// TwinCAT 3 PLC project TFM
// ProgramVersion: 3.1.4024.0
// libraries:
//   Tc2_Standard, * (Beckhoff Automation GmbH)
//   Tc2_System, * (Beckhoff Automation GmbH)
//   Tc2_Utilities, * (Beckhoff Automation GmbH)
//   Tc3_Module, * (Beckhoff Automation GmbH)
//   VisuDialogs, * (System)
//   VisuSymbols,3.5.10.0,System
// project tree:
//   DUTs/ DUT_Guardado_Almacen.TcDUT (not stored), DUT_Input.TcDUT
//   / GlobalTextList.TcGTLO, PlcTask.TcTTO (not stored), Visualization Manager.TcVMO (not stored)
//   GVLs/ GVL.TcGVL
//   POUs/Almacén/ FB_Visibilidad.TcPOU (not stored), FUN_get_Posicion_Libre_Array.TcPOU (not stored), FUN_get_Posicion_Ocupada_Array.TcPOU, POU_Almacen.TcPOU, POU_Cruce_Almacen.TcPOU, POU_Linea_Almacen.TcPOU
//   POUs/Control funcionalidad/ Contadores_Control_Lineas.TcPOU, FB_Control_Estacion.TcPOU, POU_Control_Estaciones.TcPOU (not stored), POU_Edges.TcPOU, POU_Parada.TcPOU (not stored), POU_Reset_Planta.TcPOU
//   POUs/Entrada y división/ Etapa1.TcPOU
//   POUs/Línea producción/ Linea_Produccion.TcPOU (not stored), POU_Pinzas.TcPOU
//   POUs/ MAIN.TcPOU (not stored)
//   POUs/Módulos/ POU_Control_Planta_1.TcPOU (not stored), POU_Funcionamiento.TcPOU (not stored), POU_Mando.TcPOU, POU_Seguridad.TcPOU
//   VISUs/Manual/ Almacen_Manual.TcVIS, Entrada_Manual.TcVIS (not stored), Linea_Almacen_Manual.TcVIS, Linea_Produccion_Azul_1.TcVIS, Linea_Produccion_Azul_2.TcVIS
//   VISUs/ Pantalla_Principal.TcVIS (not stored), HMI.TcVIS
// real-time tasks:
//   TASK PlcTask: cycle T#10ms, priority 20, ADS port 350

// ---- DUTs/DUT_Input.TcDUT
TYPE DUT_Input :
STRUCT
	Max_Capas_Apiladas_Azul  : INT := 2; 	  // Cantidad de capas a apilar en el paletizador	
	Max_Capas_Apiladas_Verde : INT := 2;	  // Cantidad de capas a apilar en el paletizador	
	Max_Capas_Apiladas_Metal : INT := 2; 	  // Cantidad de capas a apilar en el paletizador
	Descartar_Pieza_Azul 	 : BOOL := FALSE; // Control de ingreso de material a la línea Azul
	Descartar_Pieza_Verde  	 : BOOL := FALSE; // Control de ingreso de material a la línea Verde
	Descartar_Pieza_Metal 	 : BOOL := FALSE; // Control de ingreso de material a la línea Metal
END_STRUCT
END_TYPE

// ---- GVLs/GVL.TcGVL
//{attribute 'qualified_only'}
VAR_GLOBAL

// LOCAL
	
	Manual : BOOL := FALSE; // Control modo manual/automático
	Marcha : BOOL := FALSE; // Control modo de operación de la planta
	
	//CONTADORES TOTALES PARA BASE DE DATOS
	
	Contador_Totales_Azul_Separadas 	 : INT := 0;  // Piezas totales azules pasadas a la linea de produccion
	Contador_Totales_Verde_Separadas 	 : INT := 0;  // Piezas totales verdes pasadas a la linea de producción
	Contador_Totales_Metal_Separadas 	 : INT := 0;  // Piezas totales metalicas pasadas a la linea de producción
	Contador_Piezas_Totales_Emitidas 	 : INT := 0;  // Piezas totales emitidas por el emisor
	Contador_Piezas_Totales_Descartadas  : INT := 0;  // Piezas totales descartadas
	Contador_Palets_Azules_Totales  	 : INT := 0;  // Palets de productos azules completados
	Contador_Palets_Verdes_Totales  	 : INT := 0;  // Palets de productos verdes completados
	Contador_Palets_Metales_Totales 	 : INT := 0;  // Palets de productos metales completados
	Pallets_Almacenados 				 : DINT := 0; // Cantidad de palets almacenados sin contar los extraidos
	Pallets_Almacenados_Retirados		 : DINT := 0; // Totalidad de palets extraidos
	Pallets_Azules_Totales_Emitidos  	 : DINT := 0; // Cantidad de palets emitidos para ser "rellenados", esta variable se usa para controlar los errores del RFID		
	Pallets_Verdes_Totales_Emitidos   	 : DINT := 0; // Cantidad de palets emitidos para ser "rellenados", esta variable se usa para controlar los errores del RFID	
	Pallets_Metalicos_Totales_Emitidos   : DINT := 0; // Cantidad de palets emitidos para ser "rellenados", esta variable se usa para controlar los errores del RFID	
	
	// CONTADORES-FLAGS PARA CONTROL DE LINEA	

	//Contador_Piezas_No_Descartadas : INT := 0; // Piezas utilizables emitidas por el emitter 1,
	Capas_Apiladas_Azul					 : INT := 0;  // Capas de cajas de producto azul apiladas en el palet
	Capas_Apiladas_Metal				 : INT := 0;  // Capas de cajas de producto verde apiladas en el palet
	Capas_Apiladas_Verde				 : INT := 0;  // Capas de cajas de producto metálico apiladas en el palet
	Contador_Piezas_Zona_Pivot_Principal : INT := 0;  // Piezas en la zona Pivot y descarte
	Contador_Pivot_Azul 				 : INT := 0;  // Piezas en la zona Pivot de la linea azul
	Contador_Pivot_Verde 				 : INT := 0;  // Piezas en la zona Pivot de la linea verde
	Contador_Pivot_Metal 				 : INT := 0;  // Piezas en la zona Pivot de la linea metal
	Contador_Manipulador_1 				 : INT := 0;  // Piezas que hay dentro de la celda del robot
	Contador_Manipulador_2				 : INT := 0;  // Piezas que hay dentro de la celda del robot
	Contador_Manipulador_3				 : INT := 0;  // Piezas que hay dentro de la celda del robot
	Contador_Manipulador_4				 : INT := 0;  // Piezas que hay dentro de la celda del robot
	Contador_Manipulador_5				 : INT := 0;  // Piezas que hay dentro de la celda del robot
	Contador_Manipulador_6				 : INT := 0;  // Piezas que hay dentro de la celda del robot
	Contador_Linea_Manipulador_1_I		 : INT := 0;  // Piezas que hay en la cinta de entrada al manipulador
	Contador_Linea_Manipulador_2_I		 : INT := 0;  // Piezas que hay en la cinta de entrada al manipulador
	Contador_Linea_Manipulador_3_I		 : INT := 0;  // Piezas que hay en la cinta de entrada al manipulador	
	Contador_Linea_Manipulador_4_I		 : INT := 0;  // Piezas que hay en la cinta de entrada al manipulador	
	Contador_Linea_Manipulador_5_I		 : INT := 0;  // Piezas que hay en la cinta de entrada al manipulador
	Contador_Linea_Manipulador_6_I		 : INT := 0;  // Piezas que hay en la cinta de entrada al manipulador	
	Contador_Linea_Principal			 : INT := 0;  // Elementos en la línea principal de entrada tras el sensor de visión
	Contador_Manipulador_1_Lid			 : INT := 0;  // Piezas que hay en la cinta de salida del manipulador	
	Contador_Manipulador_2_Lid			 : INT := 0;  // Piezas que hay en la cinta de salida del manipulador	
	Contador_Manipulador_3_Lid			 : INT := 0;  // Piezas que hay en la cinta de salida del manipulador
	Contador_Manipulador_1_Base			 : INT := 0;  // Piezas que hay en la cinta de salida del manipulador
	Contador_Manipulador_2_Base			 : INT := 0;  // Piezas que hay en la cinta de salida del manipulador
	Contador_Manipulador_3_Base 		 : INT := 0;  // Piezas que hay en la cinta de salida del manipulador
	Contador_Box_Azul					 : INT := 0;  // Cajas de producto azul entrando al paletizado
	Contador_Box_Verde					 : INT := 0;  // Cajas de producto verde entrando al paletizado
	Contador_Box_Metal 					 : INT := 0;  // Cajas de producto metálico entrando al paletizado
	Contador_Palets_Azules   			 : INT := 0;  // Palets de producto azul en el primer tramo de rodillos	
	Contador_Palets_Verdes				 : INT := 0;  // Palets de producto verde en el primer tramo de rodillos	
	Contador_Palets_Metal				 : INT := 0;  // Palets de producto metálico en el primer tramo de rodillos
	Contador_Linea_Cruce_1				 : INT := 0;  // Palets que hay entre los dos cruces de rodillos
	Contador_Linea_Cruce_2				 : INT := 0;  // Palets entre el último cruce y el almacen	
	Linea_Salida_Libre_2				 : BOOL := TRUE; // Control de cinta de salida para el paletizado de laínea verde, si la línea de salida no está libre, no puede sacar el palet
	Linea_Salida_Libre_3				 : BOOL := TRUE; // Control de cinta de salida para el paletizado de la línea metálica, si la línea de salida no está libre, no puede sacar el palet

	// VARIABLES PARA CONTROLAR ACCIONES	
	
	Sacar_Palet_1 			: BOOL := FALSE; // Para saber si el palet de producto azul del paletizador tiene via libre para ser pasado a los rodillos camino al almacen
	Sacar_Palet_2 			: BOOL := FALSE; // Para saber si el palet de producto verde del paletizador tiene via libre para ser pasado a los rodillos camino al almacen
	Sacar_Palet_3			: BOOL := FALSE; // Para saber si el palet de producto metálico  paletizador tiene via libre para ser pasado a los rodillos camino al almacen
	Error_RFID_1 			: BOOL := FALSE; // Variable que guarda si ha habido error a la hora de escribir información en un palet en la línea azul	
	Error_RFID_2 			: BOOL := FALSE; // Variable que guarda si ha habido error a la hora de escribir información en un palet en la línea verde
	Error_RFID_3 			: BOOL := FALSE; // Variable que guarda si ha habido error a la hora de escribir información en un palet en la línea metálica
	Error_RFID_Almacen 		: BOOL := FALSE; // Variable que guarda si ha habido error a la hora de leer información en un palet a almacenar
	Control_TAPP_A 			: BOOL := FALSE; // En base a la botonera de control y los sensores de puerta, se permite el movimiento o no del Pick&Place de la línea azul
	Control_TAPP_V 			: BOOL := FALSE; // En base a la botonera de control y los sensores de puerta, se permite el movimiento o no del Pick&Place de la línea verde
	Control_TAPP_M 			: BOOL := FALSE; // En base a la botonera de control y los sensores de puerta, se permite el movimiento o no del Pick&Place de la línea metálica
	Control_Paletizador_A 	: BOOL := FALSE; // En base a la botonera de control y los sensores de puerta, se permite el movimiento o no del paletizador de la línea azul
	Control_Paletizador_V 	: BOOL := FALSE; // En base a la botonera de control y los sensores de puerta, se permite el movimiento o no del paletizador de la línea verde
	Control_Paletizador_M 	: BOOL := FALSE; // En base a la botonera de control y los sensores de puerta, se permite el movimiento o no del paletizador de la línea metálica
	Control_Almacen 		: BOOL := FALSE; // En base a la botonera de control y los sensores de puerta, se permite el movimiento o no de la grúa del alamcén
	Reset					: BOOL := FALSE; // Variable para resetear los contadores
	
	//ESTADOS	
	Estado_Pick_Place_1 	: INT  := 0; // Estado del Pick&Place de la línea azul
	Estado_Palletizer_1 	: INT  := 0; // Estado del Pick&Place de la línea verde
	Estado_Pick_Place_2 	: INT  := 0; // Estado del Pick&Place de la línea metálica
	Estado_Palletizer_2 	: INT  := 0; // Estado del paletizador de la línea azul
	Estado_Pick_Place_3 	: INT  := 0; // Estado del paletizador de la línea verde
	Estado_Palletizer_3 	: INT  := 0; // Estado del paletizador de la línea metálica	
	Estado_Almacen_I 		: INT  := 0; // Estado de la grúa en modo almacenamiento
	Estado_Almacen_O 		: INT  := 1; // Estado de la grúa en modo extracción
	
	// ALMACEN
	
	ContadorPalets			: INT := 0; 							// Contador de palets del Almacen en base a la selección del display
	Retirada_Start			: BOOL := FALSE; 						// Guarda la pulsación del botón start para extraer del almacen
	Clasificados 			: ARRAY[0..53] OF DUT_Guardado_Almacen; // Estanteria: 0 (posicion libre), 1 (id blue raw material), 4 (id green raw material), 7 (id metal raw material)
	Input					: ARRAY[0..0] OF DUT_Input; 			// Variables de entrada para controlar la funcionalidad del flujo.

// --------------------------- ENTRADAS ---------------------------

// Etapa Entrada 

	{attribute 'OPC.UA.DA' := '1'}
	Diffuse_Sensor_0 AT %I* : BOOL;
	{attribute 'OPC.UA.DA' := '1'}
	Diffuse_Sensor_1 AT %I* : BOOL;
	{attribute 'OPC.UA.DA' := '1'} 
	Diffuse_Sensor_2 AT %I* : BOOL;
	{attribute 'OPC.UA.DA' := '1'} 
	Diffuse_Sensor_3 AT %I* : BOOL;
	{attribute 'OPC.UA.DA' := '1'} 
	Diffuse_Sensor_4 AT %I* : BOOL;
	{attribute 'OPC.UA.DA' := '1'} 
	Diffuse_Sensor_5 AT %I* : BOOL;
	{attribute 'OPC.UA.DA' := '1'} 
	Diffuse_Sensor_8 AT %I* : BOOL;
	{attribute 'OPC.UA.DA' := '1'} 
	Diffuse_Sensor_9 AT %I* : BOOL;
	{attribute 'OPC.UA.DA' := '1'} 
	Diffuse_Sensor_12 AT %I* : BOOL;
	{attribute 'OPC.UA.DA' := '1'} 
	Emergency_Stop_2 AT %I* : BOOL;
	{attribute 'OPC.UA.DA' := '1'} 	
	Pusher_1_Front_Limit AT %I* : BOOL;
	{attribute 'OPC.UA.DA' := '1'} 
	Pusher_2_Front_Limit AT %I* : BOOL;
	{attribute 'OPC.UA.DA' := '1'} 
	Pusher_3_Front_Limit AT %I* : BOOL;	
	{attribute 'OPC.UA.DA' := '1'} 
	Reset_Button_2: BOOL;
	{attribute 'OPC.UA.DA' := '1'} 
	Start_Button_2 AT %I* : BOOL;
	{attribute 'OPC.UA.DA' := '1'} 
	Stop_Button_2 AT %I* : BOOL;
	

// Linea Producción 1 
	
	{attribute 'OPC.UA.DA' := '1'} 
	Diffuse_Sensor_15 AT %I* : BOOL;
	{attribute 'OPC.UA.DA' := '1'} 
	Diffuse_Sensor_16 AT %I* : BOOL;	
	{attribute 'OPC.UA.DA' := '1'} 
	Diffuse_Sensor_45 AT %I* : BOOL;
	{attribute 'OPC.UA.DA' := '1'} 
	Diffuse_Sensor_46 AT %I* : BOOL;
	{attribute 'OPC.UA.DA' := '1'} 
	Emergency_Stop_3 AT %I* : BOOL;
	{attribute 'OPC.UA.DA' := '1'}
	Emergency_Stop_4 AT %I* : BOOL;
	//{attribute 'OPC.UA.DA' := '1'} 
	Reset_Button_3 AT %I* : BOOL;
	//{attribute 'OPC.UA.DA' := '1'} 
	Reset_Button_4 AT %I* : BOOL;	
	//{attribute 'OPC.UA.DA' := '1'} 
	Safety_Door_1 AT %I* : BOOL;
	//{attribute 'OPC.UA.DA' := '1'} 
	Safety_Door_2 AT %I* : BOOL;
	//{attribute 'OPC.UA.DA' := '1'} 
	Safety_Door_3 AT %I* : BOOL;
	//{attribute 'OPC.UA.DA' := '1'} 
	Safety_Door_4 AT %I* : BOOL;
	//{attribute 'OPC.UA.DA' := '1'} 
	Start_Button_3 AT %I* : BOOL;
	//{attribute 'OPC.UA.DA' := '1'} 
	Stop_Button_3 AT %I* : BOOL;
	//{attribute 'OPC.UA.DA' := '1'} //Comentar
	Start_Button_6 AT %I* : BOOL;
	//{attribute 'OPC.UA.DA' := '1'} //Comentar
	Stop_Button_6 AT %I* : BOOL;
	
	
	//Función
	
	{attribute 'OPC.UA.DA' := '1'} 
	Diffuse_Sensor_6 AT %I* : BOOL;
	{attribute 'OPC.UA.DA' := '1'} 
	Diffuse_Sensor_7 AT %I* : BOOL;
	{attribute 'OPC.UA.DA' := '1'} 
	Diffuse_Sensor_17 AT %I* : BOOL;	
	{attribute 'OPC.UA.DA' := '1'} 
	Diffuse_Sensor_18 AT %I* : BOOL;	
	{attribute 'OPC.UA.DA' := '1'} 
	Diffuse_Sensor_19 AT %I* : BOOL;	
	{attribute 'OPC.UA.DA' := '1'} 
	Diffuse_Sensor_20 AT %I* : BOOL;
	{attribute 'OPC.UA.DA' := '1'} 
	Diffuse_Sensor_21 AT %I* : BOOL;
	{attribute 'OPC.UA.DA' := '1'} 
	Diffuse_Sensor_22 AT %I* : BOOL;
	{attribute 'OPC.UA.DA' := '1'}  // Comentar
	Palletizer_1_Clamped AT %I* : BOOL;	
	{attribute 'OPC.UA.DA' := '1'}  // Comentar
	Palletizer_1_Plate_Limit AT %I* : BOOL;	
	{attribute 'OPC.UA.DA' := '1'}  // Comentar
	Palletizer_1_Pusher_Limit AT %I* : BOOL;
	{attribute 'OPC.UA.DA' := '1'}  // Comentar
	Palletizer_1_Elevator_Back_Limit AT %I* : BOOL;	
	{attribute 'OPC.UA.DA' := '1'}  // Comentar
	Palletizer_1_Elevator_Front_Limit AT %I* : BOOL;	
	{attribute 'OPC.UA.DA' := '1'}  // Comentar
	Palletizer_1_Elevator_Moving AT %I* : BOOL;	
	{attribute 'OPC.UA.DA' := '1'}  // Comentar
	RFID_Reader_1_Status AT %I* : DINT;	
	{attribute 'OPC.UA.DA' := '1'}  // Comentar
	RFID_Reader_1_Command_ID AT %I* : DINT;	
	//{attribute 'OPC.UA.DA' := '1'} 
	Right_Positioner_1_Clamped AT %I* : BOOL;
	{attribute 'OPC.UA.DA' := '1'}  // Comentar
	Right_Positioner_2_Clamped AT %I* : BOOL;
	{attribute 'OPC.UA.DA' := '1'}  // Comentar
	Right_Positioner_2_Limit AT %I* : BOOL;	
	{attribute 'OPC.UA.DA' := '1'}  // Comentar
	Two_Axis_Pick_Place_1_Detected AT %I* : BOOL;	
	{attribute 'OPC.UA.DA' := '1'}  // Comentar
	Two_Axis_Pick_Place_1_MovingX AT %I* : BOOL;
	{attribute 'OPC.UA.DA' := '1'}  // Comentar
	Two_Axis_Pick_Place_1_MovingZ AT %I* : BOOL;
	
	
// Línea Producción 2	
	
	{attribute 'OPC.UA.DA' := '1'} 
	Diffuse_Sensor_23 AT %I* : BOOL;
	{attribute 'OPC.UA.DA' := '1'} 
	Diffuse_Sensor_24 AT %I* : BOOL;
	{attribute 'OPC.UA.DA' := '1'} 
	Diffuse_Sensor_47 AT %I* : BOOL;
	{attribute 'OPC.UA.DA' := '1'} 
	Diffuse_Sensor_48 AT %I* : BOOL;
	{attribute 'OPC.UA.DA' := '1'}
	Emergency_Stop_5 AT %I* : BOOL;
	{attribute 'OPC.UA.DA' := '1'}
	Emergency_Stop_6 AT %I* : BOOL;
	//{attribute 'OPC.UA.DA' := '1'} 
	Reset_Button_5 AT %I* : BOOL;
	{attribute 'OPC.UA.DA' := '1'} 
	Reset_Button_6 AT %I* : BOOL;
	//{attribute 'OPC.UA.DA' := '1'} //Comentar
	Safety_Door_5 AT %I* : BOOL;
	//{attribute 'OPC.UA.DA' := '1'} //Comentar
	Safety_Door_6 AT %I* : BOOL;
	//{attribute 'OPC.UA.DA' := '1'} //Comentar
	Safety_Door_7 AT %I* : BOOL;
	//{attribute 'OPC.UA.DA' := '1'} //Comentar
	Safety_Door_8 AT %I* : BOOL;
	//{attribute 'OPC.UA.DA' := '1'} 
	Start_Button_4 AT %I* : BOOL;
	//{attribute 'OPC.UA.DA' := '1'} 
	Stop_Button_4 AT %I* : BOOL;
	//{attribute 'OPC.UA.DA' := '1'} //Comentar
	Start_Button_7 AT %I* : BOOL;
	//{attribute 'OPC.UA.DA' := '1'} //Comentar
	Stop_Button_7 AT %I* : BOOL;
	
	
	//Función
	
	{attribute 'OPC.UA.DA' := '1'} 
	Diffuse_Sensor_10 AT %I* : BOOL;
	{attribute 'OPC.UA.DA' := '1'} 
	Diffuse_Sensor_11 AT %I* : BOOL;
	{attribute 'OPC.UA.DA' := '1'} 
	Diffuse_Sensor_25 AT %I* : BOOL;
	{attribute 'OPC.UA.DA' := '1'} 
	Diffuse_Sensor_26 AT %I* : BOOL;
	{attribute 'OPC.UA.DA' := '1'} 
	Diffuse_Sensor_27 AT %I* : BOOL;
	{attribute 'OPC.UA.DA' := '1'} 
	Diffuse_Sensor_28 AT %I* : BOOL;
	{attribute 'OPC.UA.DA' := '1'} 
	Diffuse_Sensor_29 AT %I* : BOOL;
	{attribute 'OPC.UA.DA' := '1'} 
	Diffuse_Sensor_30 AT %I* : BOOL;
	//{attribute 'OPC.UA.DA' := '1'} // Comentar
	Palletizer_2_Clamped AT %I* : BOOL;	
	//{attribute 'OPC.UA.DA' := '1'}  // Comentar
	Palletizer_2_Plate_Limit AT %I* : BOOL;	
	//{attribute 'OPC.UA.DA' := '1'}  // Comentar
	Palletizer_2_Pusher_Limit AT %I* : BOOL;
	//{attribute 'OPC.UA.DA' := '1'}  // Comentar
	Palletizer_2_Elevator_Back_Limit AT %I* : BOOL;	
	//{attribute 'OPC.UA.DA' := '1'}  // Comentar
	Palletizer_2_Elevator_Front_Limit AT %I* : BOOL;	
	//{attribute 'OPC.UA.DA' := '1'}  // Comentar
	Palletizer_2_Elevator_Moving AT %I* : BOOL;
	//{attribute 'OPC.UA.DA' := '1'}  // Comentar
	RFID_Reader_2_Status AT %I* : DINT;	
	//{attribute 'OPC.UA.DA' := '1'}
	RFID_Reader_2_Command_ID AT %I* : DINT;
	//{attribute 'OPC.UA.DA' := '1'}  // Comentar
	Right_Positioner_3_Clamped AT %I* : BOOL;	
	//{attribute 'OPC.UA.DA' := '1'}  // Comentar
	Right_Positioner_4_Clamped AT %I* : BOOL;
	//{attribute 'OPC.UA.DA' := '1'}  // Comentar
	Right_Positioner_4_Limit AT %I* : BOOL;
	//{attribute 'OPC.UA.DA' := '1'}  // Comentar
	Two_Axis_Pick_Place_2_Detected AT %I* : BOOL;
	//{attribute 'OPC.UA.DA' := '1'}  // Comentar
	Two_Axis_Pick_Place_2_MovingX AT %I* : BOOL;
	//{attribute 'OPC.UA.DA' := '1'}  // Comentar
	Two_Axis_Pick_Place_2_MovingZ AT %I* : BOOL;
	

// Línea Producción 3

	{attribute 'OPC.UA.DA' := '1'} 
	Diffuse_Sensor_31 AT %I* : BOOL;
	{attribute 'OPC.UA.DA' := '1'} 
	Diffuse_Sensor_32 AT %I* : BOOL;
	{attribute 'OPC.UA.DA' := '1'} 
	Diffuse_Sensor_49 AT %I* : BOOL;
	{attribute 'OPC.UA.DA' := '1'} 
	Diffuse_Sensor_50 AT %I* : BOOL;	
	{attribute 'OPC.UA.DA' := '1'}
	Emergency_Stop_7 AT %I* : BOOL;
	{attribute 'OPC.UA.DA' := '1'}
	Emergency_Stop_8 AT %I* : BOOL;
	//{attribute 'OPC.UA.DA' := '1'} 
	Reset_Button_7 AT %I* : BOOL;
	//{attribute 'OPC.UA.DA' := '1'} 
	Reset_Button_8 AT %I* : BOOL;
	//{attribute 'OPC.UA.DA' := '1'} //Comentar
	Safety_Door_9 AT %I* : BOOL;
	//{attribute 'OPC.UA.DA' := '1'} //Comentar
	Safety_Door_10 AT %I* : BOOL;
	//{attribute 'OPC.UA.DA' := '1'} //Comentar
	Safety_Door_11 AT %I* : BOOL;
	//{attribute 'OPC.UA.DA' := '1'} //Comentar
	Safety_Door_12 AT %I* : BOOL;
	//{attribute 'OPC.UA.DA' := '1'} //Comentar
	Start_Button_5 AT %I* : BOOL;
	//{attribute 'OPC.UA.DA' := '1'} //Comentar
	Stop_Button_5 AT %I* : BOOL;
	//{attribute 'OPC.UA.DA' := '1'} //Comentar
	Start_Button_8 AT %I* : BOOL;
	//{attribute 'OPC.UA.DA' := '1'} //Comentar
	Stop_Button_8 AT %I* : BOOL;
	
	
	//Función
	
	{attribute 'OPC.UA.DA' := '1'} 
	Diffuse_Sensor_13 AT %I* : BOOL;
	{attribute 'OPC.UA.DA' := '1'} 
	Diffuse_Sensor_14 AT %I* : BOOL;
	{attribute 'OPC.UA.DA' := '1'} 
	Diffuse_Sensor_33 AT %I* : BOOL;
	{attribute 'OPC.UA.DA' := '1'} 
	Diffuse_Sensor_34 AT %I* : BOOL;
	{attribute 'OPC.UA.DA' := '1'} 
	Diffuse_Sensor_35 AT %I* : BOOL;
	{attribute 'OPC.UA.DA' := '1'} 
	Diffuse_Sensor_36 AT %I* : BOOL;
	{attribute 'OPC.UA.DA' := '1'} 
	Diffuse_Sensor_37 AT %I* : BOOL;
	{attribute 'OPC.UA.DA' := '1'} 
	Diffuse_Sensor_38 AT %I* : BOOL;
	//{attribute 'OPC.UA.DA' := '1'}  // Comentar
	Palletizer_3_Clamped AT %I* : BOOL;	
	//{attribute 'OPC.UA.DA' := '1'}  // Comentar
	Palletizer_3_Plate_Limit AT %I* : BOOL;
	//{attribute 'OPC.UA.DA' := '1'}  // Comentar
	Palletizer_3_Pusher_Limit AT %I* : BOOL;
	//{attribute 'OPC.UA.DA' := '1'}  // Comentar
	Palletizer_3_Elevator_Back_Limit AT %I* : BOOL;
	//{attribute 'OPC.UA.DA' := '1'}  // Comentar
	Palletizer_3_Elevator_Front_Limit AT %I* : BOOL;
	//{attribute 'OPC.UA.DA' := '1'}  // Comentar
	Palletizer_3_Elevator_Moving AT %I* : BOOL;	
	//{attribute 'OPC.UA.DA' := '1'}  // Comentar
	RFID_Reader_3_Status AT %I* : DINT;	
	//{attribute 'OPC.UA.DA' := '1'}  // Comentar
	RFID_Reader_3_Command_ID AT %I* : DINT;	
	//{attribute 'OPC.UA.DA' := '1'}  // Comentar
	Right_Positioner_5_Clamped AT %I* : BOOL;
	//{attribute 'OPC.UA.DA' := '1'}  // Comentar
	Right_Positioner_6_Clamped AT %I* : BOOL;
	//{attribute 'OPC.UA.DA' := '1'}  // Comentar
	Right_Positioner_6_Limit AT %I* : BOOL;
	//{attribute 'OPC.UA.DA' := '1'}  // Comentar
	Two_Axis_Pick_Place_3_Detected AT %I* : BOOL;
	//{attribute 'OPC.UA.DA' := '1'}  // Comentar
	Two_Axis_Pick_Place_3_MovingX AT %I* : BOOL;
	//{attribute 'OPC.UA.DA' := '1'}  // Comentar
	Two_Axis_Pick_Place_3_MovingZ AT %I* : BOOL;
	
	
//Línea Almacén
	
	{attribute 'OPC.UA.DA' := '1'} 
	Diffuse_Sensor_39 AT %I* : BOOL;
	{attribute 'OPC.UA.DA' := '1'} 
	Diffuse_Sensor_40 AT %I* : BOOL;
	{attribute 'OPC.UA.DA' := '1'} 
	Diffuse_Sensor_41 AT %I* : BOOL;
	{attribute 'OPC.UA.DA' := '1'} 
	Diffuse_Sensor_42 AT %I* : BOOL;
	{attribute 'OPC.UA.DA' := '1'} 
	Diffuse_Sensor_43 AT %I* : BOOL;
	{attribute 'OPC.UA.DA' := '1'} 
	Diffuse_Sensor_44 AT %I* : BOOL;
	{attribute 'OPC.UA.DA' := '1'} 
	Emergency_Stop_1 AT %I* : BOOL;
	{attribute 'OPC.UA.DA' := '1'}
	Emergency_Stop_9 AT %I* : BOOL;
	{attribute 'OPC.UA.DA' := '1'} 
	Stacker_Crane_1_Left_Limit AT %I* : BOOL;	
	{attribute 'OPC.UA.DA' := '1'} 
	Stacker_Crane_1_Middle_Limit AT %I* : BOOL;
	{attribute 'OPC.UA.DA' := '1'} 
	Stacker_Crane_1_Moving_X AT %I* : BOOL;
	{attribute 'OPC.UA.DA' := '1'} 
	Stacker_Crane_1_Moving_Z AT %I* : BOOL;
	{attribute 'OPC.UA.DA' := '1'} 
	Stacker_Crane_1_Right_Limit AT %I* : BOOL;
	{attribute 'OPC.UA.DA' := '1'} 
	Turnable_1_Back_Limit AT %I* : BOOL;
	{attribute 'OPC.UA.DA' := '1'} 
	Turnable_1_Limit_0 AT %I* : BOOL;
	{attribute 'OPC.UA.DA' := '1'} 
	Turnable_1_Limit_90 AT %I* : BOOL;
	{attribute 'OPC.UA.DA' := '1'} 
	Turnable_2_Back_Limit AT %I* : BOOL;
	{attribute 'OPC.UA.DA' := '1'} 
	Turnable_2_Limit_0 AT %I* : BOOL;
	{attribute 'OPC.UA.DA' := '1'} 
	Turnable_2_Limit_90 AT %I* : BOOL;		
	{attribute 'OPC.UA.DA' := '1'} 
	Vision_Sensor_1 AT %I* : DINT;
	{attribute 'OPC.UA.DA' := '1'} 
	Reset_Button_1 AT %I* : BOOL;
	//{attribute 'OPC.UA.DA' := '1'} 
	Reset_Button_9 AT %I* : BOOL;
	{attribute 'OPC.UA.DA' := '1'} 
	Retroreflective_Sensor_1 AT %I* : BOOL;	
	{attribute 'OPC.UA.DA' := '1'} 
	Retroreflective_Sensor_2 AT %I* : BOOL;		
	{attribute 'OPC.UA.DA' := '1'} 
	RFID_Reader_4_Read_Data AT %I* : DINT := 1;				
	{attribute 'OPC.UA.DA' := '1'} 
	RFID_Reader_4_Status AT %I* : DINT;		
	{attribute 'OPC.UA.DA' := '1'} 
	RFID_Reader_4_Command_ID AT %I* : DINT;
	{attribute 'OPC.UA.DA' := '1'} 
	Safety_Door_13 AT %I* : BOOL;
	{attribute 'OPC.UA.DA' := '1'} 
	Safety_Door_14 AT %I* : BOOL;
	{attribute 'OPC.UA.DA' := '1'} 
	Safety_Door_15 AT %I* : BOOL;
	{attribute 'OPC.UA.DA' := '1'} 
	Start_Button_1 AT %I* : BOOL;
	{attribute 'OPC.UA.DA' := '1'} 
	Stop_Button_1 AT %I* : BOOL;
	{attribute 'OPC.UA.DA' := '1'} //Comentar
	Start_Button_9 AT %I* : BOOL;
	{attribute 'OPC.UA.DA' := '1'} //Comentar
	Stop_Button_9 AT %I* : BOOL;
	{attribute 'OPC.UA.DA' := '1'} 
	Selector1_State_1 AT %I* : BOOL;
	{attribute 'OPC.UA.DA' := '1'} 
	Selector1_State_2 AT %I* : BOOL;
	//{attribute 'OPC.UA.DA' := '1'} 
	Turnable_1_Front_Limit AT %I* : BOOL;
	//{attribute 'OPC.UA.DA' := '1'} 
	Turnable_2_Front_Limit AT %I* : BOOL;

	
//Exclusivo HMI

	//{attribute 'OPC.UA.DA' := '1'} 
	Machining_Center_1_IsBusy AT %I* : BOOL;
	//{attribute 'OPC.UA.DA' := '1'} 
	Machining_Center_1_Error AT %I* : BOOL;
	//{attribute 'OPC.UA.DA' := '1'} 
	Machining_Center_1_Opened AT %I* : BOOL;
	//{attribute 'OPC.UA.DA' := '1'} 
	Machining_Center_1_Progress AT %I* : REAL;
	//{attribute 'OPC.UA.DA' := '1'} 
	Machining_Center_2_IsBusy AT %I* : BOOL;
	//{attribute 'OPC.UA.DA' := '1'} 
	Machining_Center_2_Error AT %I* : BOOL;
	//{attribute 'OPC.UA.DA' := '1'} 
	Machining_Center_2_Opened AT %I* : BOOL;
	//{attribute 'OPC.UA.DA' := '1'} 
	Machining_Center_2_Progress AT %I* : REAL;	
	// {attribute 'OPC.UA.DA' := '1'
	Machining_Center_3_IsBusy AT %I* : BOOL;
	// {attribute 'OPC.UA.DA' := '1'}
	Machining_Center_3_Error AT %I* : BOOL;
	// {attribute 'OPC.UA.DA' := '1'} 
	Machining_Center_3_Opened AT %I* : BOOL;
	// {attribute 'OPC.UA.DA' := '1'}
	Machining_Center_3_Progress AT %I* : REAL;
	// {attribute 'OPC.UA.DA' := '1'}
	Machining_Center_4_IsBusy AT %I* : BOOL;
	// {attribute 'OPC.UA.DA' := '1'}
	Machining_Center_4_Error AT %I* : BOOL;
	// {attribute 'OPC.UA.DA' := '1'}
	Machining_Center_4_Opened AT %I* : BOOL;
	// {attribute 'OPC.UA.DA' := '1'}
	Machining_Center_4_Progress AT %I* : REAL;
	// {attribute 'OPC.UA.DA' := '1'}  
	Machining_Center_5_IsBusy AT %I* : BOOL;
	// {attribute 'OPC.UA.DA' := '1'}  
	Machining_Center_5_Error AT %I* : BOOL;
	// {attribute 'OPC.UA.DA' := '1'}  
	Machining_Center_5_Opened AT %I* : BOOL;
	// {attribute 'OPC.UA.DA' := '1'}  
	Machining_Center_5_Progress AT %I* : REAL;
	// {attribute 'OPC.UA.DA' := '1'}  
	Machining_Center_6_IsBusy AT %I* : BOOL;
	// {attribute 'OPC.UA.DA' := '1'}  
	Machining_Center_6_Error AT %I* : BOOL;
	// {attribute 'OPC.UA.DA' := '1'}  
	Machining_Center_6_Opened AT %I* : BOOL;
	// {attribute 'OPC.UA.DA' := '1'} 
	Machining_Center_6_Progress AT %I* : REAL;
	//{attribute 'OPC.UA.DA' := '1'} 	
	Pusher_1_Back_Limit AT %I* : BOOL;
	//{attribute 'OPC.UA.DA' := '1'} 
	Pusher_2_Back_Limit AT %I* : BOOL;
	//{attribute 'OPC.UA.DA' := '1'} 
	Pusher_3_Back_Limit AT %I* : BOOL;	
	//{attribute 'OPC.UA.DA' := '1'}  
	RFID_Reader_1_Read_Data AT %I* : DINT;	
	//{attribute 'OPC.UA.DA' := '1'}  
	RFID_Reader_2_Read_Data  AT %I* : DINT;	
	//{attribute 'OPC.UA.DA' := '1'}  
	RFID_Reader_3_Read_Data  AT %I* : DINT;		
	//{attribute 'OPC.UA.DA' := '1'}
	Right_Positioner_1_Limit AT %I* : BOOL;	
	//{attribute 'OPC.UA.DA' := '1'}
	Right_Positioner_3_Limit AT %I* : BOOL;	
	//{attribute 'OPC.UA.DA' := '1'}
	Right_Positioner_5_Limit AT %I* : BOOL;
	//{attribute 'OPC.UA.DA' := '1'} 
	Two_Axis_Pick_Place_1_Gripper_Rotating AT %I* : BOOL;
	//{attribute 'OPC.UA.DA' := '1'}
	Two_Axis_Pick_Place_1_Rotating AT %I* : BOOL;
	
	
			
	
	
	

// --------------------------- SALIDAS ---------------------------	

	{attribute 'OPC.UA.DA' := '1'} 
	Alarm_Siren AT %Q* : BOOL;
	{attribute 'OPC.UA.DA' := '1'} 
	Warning_Light AT %Q* : BOOL;
	{attribute 'OPC.UA.DA' := '1'} 
	Factory_IO_Pause AT %Q* : BOOL;
	{attribute 'OPC.UA.DA' := '1'} 
	Factory_IO_Reset AT %Q* : BOOL;
	
//Etapa Entrada

	{attribute 'OPC.UA.DA' := '1'} 
	Belt_Conveyor_2m_1 AT %Q* : DINT;		
	{attribute 'OPC.UA.DA' := '1'} 
	Belt_Conveyor_4m_1 AT %Q* : BOOL;
	{attribute 'OPC.UA.DA' := '1'} 
	Belt_Conveyor_6m_1 AT %Q* : BOOL;
	{attribute 'OPC.UA.DA' := '1'} 
	Belt_Conveyor_6m_4 AT %Q* : BOOL;
	{attribute 'OPC.UA.DA' := '1'} 
	Belt_Conveyor_6m_5 AT %Q* : BOOL;
	{attribute 'OPC.UA.DA' := '1'} 
	Emitter_1 AT %Q* : BOOL;
	{attribute 'OPC.UA.DA' := '1'} 
	Pivot_Arm_Sorter_1_Belt_mas AT %Q* : BOOL;
	{attribute 'OPC.UA.DA' := '1'} 
	Pivot_Arm_Sorter_1_Belt_menos AT %Q* : BOOL;
	{attribute 'OPC.UA.DA' := '1'} 
	Pusher_1 AT %Q* : BOOL;
	{attribute 'OPC.UA.DA' := '1'} 
	Pusher_2 AT %Q* : BOOL;
	{attribute 'OPC.UA.DA' := '1'} 
	Pusher_3 AT %Q* : BOOL;
	//{attribute 'OPC.UA.DA' := '1'} 
	Reset_Button_2_Light AT %Q* : BOOL;		
	//{attribute 'OPC.UA.DA' := '1'} 
	Start_Button_2_Light AT %Q* : BOOL;	
	//{attribute 'OPC.UA.DA' := '1'} 
	Stop_Button_2_Light AT %Q* : BOOL;
	
	
//Línea Producción 1
	
	{attribute 'OPC.UA.DA' := '1'} 
	Belt_Conveyor_2m_3 AT %Q* : BOOL;
	{attribute 'OPC.UA.DA' := '1'} 
	Belt_Conveyor_2m_4 AT %Q* : BOOL;
	{attribute 'OPC.UA.DA' := '1'} 
	Belt_Conveyor_2m_5 AT %Q* : BOOL;
	{attribute 'OPC.UA.DA' := '1'} 
	Belt_Conveyor_2m_6 AT %Q* : BOOL;	
	{attribute 'OPC.UA.DA' := '1'} 
	Belt_Conveyor_6m_2 AT %Q* : BOOL;
	{attribute 'OPC.UA.DA' := '1'} 
	Curved_Belt_Conveyor_1_CW AT %Q* : BOOL;
	{attribute 'OPC.UA.DA' := '1'} 
	Curved_Belt_Conveyor_1_CCW AT %Q* : BOOL;
	{attribute 'OPC.UA.DA' := '1'}  // Comentar
	Emitter_2 AT %Q* : BOOL := TRUE;
	{attribute 'OPC.UA.DA' := '1'} 
	Machining_Center_1_Produce_Lids AT %Q* : BOOL := TRUE;
	//{attribute 'OPC.UA.DA' := '1'} 
	Machining_Center_1_Start AT %Q* : BOOL;
	//{attribute 'OPC.UA.DA' := '1'} 
	Machine_Center_1_Stop  AT %Q* : BOOL ;	
	//{attribute 'OPC.UA.DA' := '1'} 
	Machine_Center_1_Reset  AT %Q* : BOOL ;
	{attribute 'OPC.UA.DA' := '1'} 
	Machining_Center_2_Produce_Lids AT %Q* : BOOL := FALSE;	
	//{attribute 'OPC.UA.DA' := '1'} 
	Machining_Center_2_Start AT %Q* : BOOL;
	//{attribute 'OPC.UA.DA' := '1'} 
	Machine_Center_2_Stop  AT %Q* : BOOL ;	
	//{attribute 'OPC.UA.DA' := '1'} 
	Machine_Center_2_Reset  AT %Q* : BOOL ;
	{attribute 'OPC.UA.DA' := '1'} 
	Pivot_Arm_Sorter_2_Belt_mas AT %Q* : BOOL;	
	//{attribute 'OPC.UA.DA' := '1'} 
	Reset_Button_3_Light AT %Q* : BOOL;	
	//{attribute 'OPC.UA.DA' := '1'} 
	Reset_Button_6_Light AT %Q* : BOOL;
	{attribute 'OPC.UA.DA' := '1'} 
	RFID_Reader_1_Command AT %Q* : DINT := 3;
	{attribute 'OPC.UA.DA' := '1'} 
	RFID_Reader_1_Write_Data AT %Q* : DINT := 1;	
	{attribute 'OPC.UA.DA' := '1'} // Comentar
	Stack_Light_1_Green AT %Q* : BOOL;	
	{attribute 'OPC.UA.DA' := '1'} // Comentar
	Stack_Light_2_Green AT %Q* : BOOL;
	{attribute 'OPC.UA.DA' := '1'} // Comentar
	Stack_Light_3_Green AT %Q* : BOOL;
	{attribute 'OPC.UA.DA' := '1'} // Comentar
	Stack_Light_4_Green AT %Q* : BOOL;	
	{attribute 'OPC.UA.DA' := '1'} // Comentar
	Stack_Light_1_Red AT %Q* : BOOL;	
	{attribute 'OPC.UA.DA' := '1'} // Comentar
	Stack_Light_2_Red AT %Q* : BOOL;
	{attribute 'OPC.UA.DA' := '1'} // Comentar
	Stack_Light_3_Red AT %Q* : BOOL;	
	{attribute 'OPC.UA.DA' := '1'} // Comentar
	Stack_Light_4_Red AT %Q* : BOOL;	
	{attribute 'OPC.UA.DA' := '1'} // Comentar
	Stack_Light_1_Yellow AT %Q* : BOOL;	
	{attribute 'OPC.UA.DA' := '1'} // Comentar
	Stack_Light_2_Yellow AT %Q* : BOOL;		
	{attribute 'OPC.UA.DA' := '1'} // Comentar
	Stack_Light_3_Yellow AT %Q* : BOOL;		
	{attribute 'OPC.UA.DA' := '1'} // Comentar
	Stack_Light_4_Yellow AT %Q* : BOOL;
	//{attribute 'OPC.UA.DA' := '1'} //comentar
	Start_Button_3_Light AT %Q* : BOOL;	
	//{attribute 'OPC.UA.DA' := '1'} 
	Start_Button_6_Light AT %Q* : BOOL;	
	//{attribute 'OPC.UA.DA' := '1'} //comentar
	Stop_Button_3_Light AT %Q* : BOOL;
	//{attribute 'OPC.UA.DA' := '1'} 
	Stop_Button_6_Light AT %Q* : BOOL;	
	
	
	//Función
	
	{attribute 'OPC.UA.DA' := '1'} 
	Belt_Conveyor_4m_4 AT %Q* : BOOL;
	{attribute 'OPC.UA.DA' := '1'} 
	Belt_Conveyor_4m_5 AT %Q* : BOOL;
	{attribute 'OPC.UA.DA' := '1'} 
	Belt_Conveyor_4m_6 AT %Q* : BOOL;
	{attribute 'OPC.UA.DA' := '1'} 
	Belt_Conveyor_4m_7 AT %Q* : BOOL;
	{attribute 'OPC.UA.DA' := '1'} 
	Belt_Conveyor_2m_13 AT %Q* : BOOL;	
	{attribute 'OPC.UA.DA' := '1'} 
	Belt_Conveyor_2m_14 AT %Q* : BOOL;	
	{attribute 'OPC.UA.DA' := '1'} 
	Belt_Conveyor_2m_15 AT %Q* : BOOL;	
	{attribute 'OPC.UA.DA' := '1'}  // Comentar
	Belt_Conveyor_Inclined_1 AT %Q* : BOOL;		
	{attribute 'OPC.UA.DA' := '1'}  // Comentar
	Emitter_5 AT %Q* : BOOL := FALSE;
	{attribute 'OPC.UA.DA' := '1'}  // Comentar
	Palletizer_1_Belt_mas AT %Q* : BOOL;
	{attribute 'OPC.UA.DA' := '1'}  // Comentar
	Palletizer_1_Chain_mas AT %Q* : BOOL;
	{attribute 'OPC.UA.DA' := '1'}  // Comentar
	Palletizer_1_Clamb AT %Q* : BOOL;	
	{attribute 'OPC.UA.DA' := '1'}  // Comentar
	Palletizer_1_Elevator_mas AT %Q* : BOOL;
	{attribute 'OPC.UA.DA' := '1'}  // Comentar
	Palletizer_1_Elevator_menos AT %Q* : BOOL;
	{attribute 'OPC.UA.DA' := '1'}  // Comentar
	Palletizer_1_Elevator_Move_Limit AT %Q* : BOOL;
	{attribute 'OPC.UA.DA' := '1'}  // Comentar
	Palletizer_1_Open_Plate AT %Q* : BOOL;
	{attribute 'OPC.UA.DA' := '1'}  // Comentar
	Palletizer_1_Push AT %Q* : BOOL;
	{attribute 'OPC.UA.DA' := '1'}  // Comentar
	Palletizer_1_Turn AT %Q* : BOOL;
	{attribute 'OPC.UA.DA' := '1'} 
	Pivot_Arm_Sorter_2_Turn AT %Q* : BOOL;
	{attribute 'OPC.UA.DA' := '1'}  // Comentar
	RFID_Reader_1_Ejecute_Comm AT %Q* : BOOL;	
	{attribute 'OPC.UA.DA' := '1'}  // Comentar
	Right_Positioner_1_Clamp AT %Q* : BOOL;
	{attribute 'OPC.UA.DA' := '1'}  // Comentar
	Right_Positioner_2_Clamp AT %Q* : BOOL;	
	{attribute 'OPC.UA.DA' := '1'}  // Comentar
	Right_Positioner_2_Raise AT %Q* : BOOL;
	{attribute 'OPC.UA.DA' := '1'} 
	Roller_Conveyor_2m_1 AT %Q* : BOOL;	
	{attribute 'OPC.UA.DA' := '1'}  // Comentar
	Two_Axis_Pick_Place_1X AT %Q* : BOOL;	
	{attribute 'OPC.UA.DA' := '1'}  // Comentar
	Two_Axis_Pick_Place_1Z AT %Q* : BOOL;	
	{attribute 'OPC.UA.DA' := '1'}  // Comentar
	Two_Axis_Pick_Place_1_Grab AT %Q* : BOOL;	
	
	
//Línea Producción 2

	{attribute 'OPC.UA.DA' := '1'} 
	Belt_Conveyor_2m_7 AT %Q* : BOOL;
	{attribute 'OPC.UA.DA' := '1'} 
	Belt_Conveyor_2m_8 AT %Q* : BOOL;
	{attribute 'OPC.UA.DA' := '1'} 
	Belt_Conveyor_2m_9 AT %Q* : BOOL;
	{attribute 'OPC.UA.DA' := '1'} 
	Belt_Conveyor_2m_10 AT %Q* : BOOL;
	{attribute 'OPC.UA.DA' := '1'} 
	Belt_Conveyor_6m_3 AT %Q* : BOOL;
	{attribute 'OPC.UA.DA' := '1'} 
	Curved_Belt_Conveyor_2_CW AT %Q* : BOOL;
	{attribute 'OPC.UA.DA' := '1'} 
	Curved_Belt_Conveyor_2_CCW AT %Q* : BOOL;
	//{attribute 'OPC.UA.DA' := '1'}  // Comentar
	Emitter_3 AT %Q* : BOOL := TRUE;
	//{attribute 'OPC.UA.DA' := '1'} 
	Machining_Center_3_Produce_Lids AT %Q* : BOOL := TRUE;
	//{attribute 'OPC.UA.DA' := '1'} 
	Machining_Center_3_Start AT %Q* : BOOL;
	//{attribute 'OPC.UA.DA' := '1'} 
	Machine_Center_3_Stop  AT %Q* : BOOL ;	
	//{attribute 'OPC.UA.DA' := '1'} 
	Machine_Center_3_Reset  AT %Q* : BOOL ;
	//{attribute 'OPC.UA.DA' := '1'} 
	Machining_Center_4_Produce_Lids AT %Q* : BOOL := FALSE;	
	//{attribute 'OPC.UA.DA' := '1'} 
	Machining_Center_4_Start AT %Q* : BOOL;
	//{attribute 'OPC.UA.DA' := '1'} 
	Machine_Center_4_Stop  AT %Q* : BOOL ;	
	//{attribute 'OPC.UA.DA' := '1'} 
	Machine_Center_4_Reset  AT %Q* : BOOL ;
	{attribute 'OPC.UA.DA' := '1'} 
	Pivot_Arm_Sorter_3_Belt_mas AT %Q* : BOOL;	
	//{attribute 'OPC.UA.DA' := '1'} 
	Reset_Button_4_Light AT %Q* : BOOL;	
	//{attribute 'OPC.UA.DA' := '1'} 
	RFID_Reader_2_Command AT %Q* : DINT := 3;
	//{attribute 'OPC.UA.DA' := '1'} 
	RFID_Reader_2_Write_Data AT %Q* : DINT := 4;
	//{attribute 'OPC.UA.DA' := '1'} 
	Reset_Button_7_Light AT %Q* : BOOL;		
	//{attribute 'OPC.UA.DA' := '1'} // Comentar
	Stack_Light_5_Green AT %Q* : BOOL;	
	//{attribute 'OPC.UA.DA' := '1'} // Comentar
	Stack_Light_6_Green AT %Q* : BOOL;
	//{attribute 'OPC.UA.DA' := '1'} // Comentar
	Stack_Light_7_Green AT %Q* : BOOL;
	//{attribute 'OPC.UA.DA' := '1'} // Comentar
	Stack_Light_8_Green AT %Q* : BOOL;	
	//{attribute 'OPC.UA.DA' := '1'} // Comentar
	Stack_Light_5_Red AT %Q* : BOOL;	
	//{attribute 'OPC.UA.DA' := '1'} // Comentar
	Stack_Light_6_Red AT %Q* : BOOL;
	//{attribute 'OPC.UA.DA' := '1'} // Comentar
	Stack_Light_7_Red AT %Q* : BOOL;	
	//{attribute 'OPC.UA.DA' := '1'} // Comentar
	Stack_Light_8_Red AT %Q* : BOOL;	
	//{attribute 'OPC.UA.DA' := '1'} // Comentar
	Stack_Light_5_Yellow AT %Q* : BOOL;	
	//{attribute 'OPC.UA.DA' := '1'} // Comentar
	Stack_Light_6_Yellow AT %Q* : BOOL;		
	//{attribute 'OPC.UA.DA' := '1'} // Comentar
	Stack_Light_7_Yellow AT %Q* : BOOL;		
	//{attribute 'OPC.UA.DA' := '1'} // Comentar
	Stack_Light_8_Yellow AT %Q* : BOOL;
	//{attribute 'OPC.UA.DA' := '1'} 
	Start_Button_4_Light AT %Q* : BOOL;
	//{attribute 'OPC.UA.DA' := '1'} 
	Start_Button_7_Light AT %Q* : BOOL;
	//{attribute 'OPC.UA.DA' := '1'} 
	Stop_Button_4_Light AT %Q* : BOOL;	
	//{attribute 'OPC.UA.DA' := '1'} 
	Stop_Button_7_Light AT %Q* : BOOL;
	
	
	//Función 
	
	{attribute 'OPC.UA.DA' := '1'} 
	Belt_Conveyor_4m_10 AT %Q* : BOOL;
	{attribute 'OPC.UA.DA' := '1'} 
	Belt_Conveyor_4m_11 AT %Q* : BOOL;
	{attribute 'OPC.UA.DA' := '1'} 
	Belt_Conveyor_2m_16 AT %Q* : BOOL;
	{attribute 'OPC.UA.DA' := '1'} 
	Belt_Conveyor_2m_17 AT %Q* : BOOL;
	{attribute 'OPC.UA.DA' := '1'} 
	Belt_Conveyor_2m_18 AT %Q* : BOOL;
	{attribute 'OPC.UA.DA' := '1'} 
	Belt_Conveyor_4m_8 AT %Q* : BOOL;
	{attribute 'OPC.UA.DA' := '1'} 
	Belt_Conveyor_4m_9 AT %Q* : BOOL;
	{attribute 'OPC.UA.DA' := '1'} 
	Belt_Conveyor_Inclined_2 AT %Q* : BOOL;	
	//{attribute 'OPC.UA.DA' := '1'}  // Comentar
	Emitter_6 AT %Q* : BOOL := FALSE;
	//{attribute 'OPC.UA.DA' := '1'}  // Comentar
	Palletizer_2_Belt_mas AT %Q* : BOOL;
	//{attribute 'OPC.UA.DA' := '1'}  // Comentar
	Palletizer_2_Chain_mas AT %Q* : BOOL;
	//{attribute 'OPC.UA.DA' := '1'}  // Comentar
	Palletizer_2_Clamb AT %Q* : BOOL;
	//{attribute 'OPC.UA.DA' := '1'}  // Comentar
	Palletizer_2_Elevator_mas AT %Q* : BOOL;
	//{attribute 'OPC.UA.DA' := '1'}  // Comentar
	Palletizer_2_Elevator_menos AT %Q* : BOOL;
	//{attribute 'OPC.UA.DA' := '1'}  // Comentar
	Palletizer_2_Elevator_Move_Limit AT %Q* : BOOL;
	//{attribute 'OPC.UA.DA' := '1'}  // Comentar
	Palletizer_2_Open_Plate AT %Q* : BOOL;
	//{attribute 'OPC.UA.DA' := '1'}  // Comentar
	Palletizer_2_Push AT %Q* : BOOL;
	//{attribute 'OPC.UA.DA' := '1'}  // Comentar
	Palletizer_2_Turn AT %Q* : BOOL;	
	{attribute 'OPC.UA.DA' := '1'} 
	Pivot_Arm_Sorter_3_Turn AT %Q* : BOOL;
	//{attribute 'OPC.UA.DA' := '1'}  // Comentar
	RFID_Reader_2_Ejecute_Comm AT %Q* : BOOL;
	//{attribute 'OPC.UA.DA' := '1'}  // Comentar
	Right_Positioner_3_Clamp AT %Q* : BOOL;
	//{attribute 'OPC.UA.DA' := '1'}  // Comentar
	Right_Positioner_4_Clamp AT %Q* : BOOL;
	//{attribute 'OPC.UA.DA' := '1'}  // Comentar
	Right_Positioner_4_Raise AT %Q* : BOOL;
	{attribute 'OPC.UA.DA' := '1'} 
	Roller_Conveyor_2m_4 AT %Q* : BOOL;
	//{attribute 'OPC.UA.DA' := '1'}  // Comentar
	Two_Axis_Pick_Place_2X AT %Q* : BOOL;
	//{attribute 'OPC.UA.DA' := '1'}  // Comentar
	Two_Axis_Pick_Place_2Z AT %Q* : BOOL;
	//{attribute 'OPC.UA.DA' := '1'}  // Comentar
	Two_Axis_Pick_Place_2_Grab AT %Q* : BOOL;	
	
	
//Línea Producción 3
	
	{attribute 'OPC.UA.DA' := '1'} 
	Belt_Conveyor_2m_2 AT %Q* : BOOL;
	{attribute 'OPC.UA.DA' := '1'} 
	Belt_Conveyor_2m_11 AT %Q* : BOOL;	
	{attribute 'OPC.UA.DA' := '1'} 
	Belt_Conveyor_2m_12 AT %Q* : BOOL;		
	{attribute 'OPC.UA.DA' := '1'} 
	Belt_Conveyor_4m_3 AT %Q* : BOOL;
	{attribute 'OPC.UA.DA' := '1'} 
	Belt_Conveyor_6m_6 AT %Q* : BOOL;	
	{attribute 'OPC.UA.DA' := '1'} 
	Curved_Belt_Conveyor_3_CW AT %Q* : BOOL;
	{attribute 'OPC.UA.DA' := '1'} 
	Curved_Belt_Conveyor_3_CCW AT %Q* : BOOL;
	//{attribute 'OPC.UA.DA' := '1'}  // Comentar
	Emitter_4 AT %Q* : BOOL := TRUE;	
	//{attribute 'OPC.UA.DA' := '1'} 
	Machining_Center_5_Produce_Lids AT %Q* : BOOL := TRUE;
	//{attribute 'OPC.UA.DA' := '1'} 
	Machining_Center_5_Start AT %Q* : BOOL;
	//{attribute 'OPC.UA.DA' := '1'} 
	Machine_Center_5_Stop  AT %Q* : BOOL ;	
	//{attribute 'OPC.UA.DA' := '1'} 
	Machine_Center_5_Reset  AT %Q* : BOOL ;
	//{attribute 'OPC.UA.DA' := '1'} 
	Machining_Center_6_Produce_Lids AT %Q* : BOOL := FALSE;	
	//{attribute 'OPC.UA.DA' := '1'} 
	Machining_Center_6_Start AT %Q* : BOOL;
	//{attribute 'OPC.UA.DA' := '1'} 
	Machine_Center_6_Stop  AT %Q* : BOOL ;	
	//{attribute 'OPC.UA.DA' := '1'} 
	Machine_Center_6_Reset  AT %Q* : BOOL ;
	{attribute 'OPC.UA.DA' := '1'} 
	Pivot_Arm_Sorter_4_Belt_mas AT %Q* : BOOL;	
	//{attribute 'OPC.UA.DA' := '1'} 
	Reset_Button_5_Light AT %Q* : BOOL;
	//{attribute 'OPC.UA.DA' := '1'} 
	Reset_Button_8_Light AT %Q* : BOOL;		
	//{attribute 'OPC.UA.DA' := '1'} 
	RFID_Reader_3_Command AT %Q* : DINT := 3;
	//{attribute 'OPC.UA.DA' := '1'} 
	RFID_Reader_3_Write_Data AT %Q* : DINT := 7;
	//{attribute 'OPC.UA.DA' := '1'} // Comentar
	Stack_Light_9_Green AT %Q* : BOOL;	
	//{attribute 'OPC.UA.DA' := '1'} // Comentar
	Stack_Light_10_Green AT %Q* : BOOL;
	//{attribute 'OPC.UA.DA' := '1'} // Comentar
	Stack_Light_11_Green AT %Q* : BOOL;
	//{attribute 'OPC.UA.DA' := '1'} // Comentar
	Stack_Light_12_Green AT %Q* : BOOL;	
	//{attribute 'OPC.UA.DA' := '1'} // Comentar
	Stack_Light_9_Red AT %Q* : BOOL;	
	//{attribute 'OPC.UA.DA' := '1'} // Comentar
	Stack_Light_10_Red AT %Q* : BOOL;
	//{attribute 'OPC.UA.DA' := '1'} // Comentar
	Stack_Light_11_Red AT %Q* : BOOL;	
	//{attribute 'OPC.UA.DA' := '1'} // Comentar
	Stack_Light_12_Red AT %Q* : BOOL;	
	//{attribute 'OPC.UA.DA' := '1'} // Comentar
	Stack_Light_9_Yellow AT %Q* : BOOL;	
	//{attribute 'OPC.UA.DA' := '1'} // Comentar
	Stack_Light_10_Yellow AT %Q* : BOOL;		
	//{attribute 'OPC.UA.DA' := '1'} // Comentar
	Stack_Light_11_Yellow AT %Q* : BOOL;		
	//{attribute 'OPC.UA.DA' := '1'} // Comentar
	Stack_Light_12_Yellow AT %Q* : BOOL;
	//{attribute 'OPC.UA.DA' := '1'} 
	Start_Button_5_Light AT %Q* : BOOL;	
	//{attribute 'OPC.UA.DA' := '1'} 
	Start_Button_8_Light AT %Q* : BOOL;	
	//{attribute 'OPC.UA.DA' := '1'} 
	Stop_Button_5_Light AT %Q* : BOOL;
	//{attribute 'OPC.UA.DA' := '1'} 
	Stop_Button_8_Light AT %Q* : BOOL;
	
	
	//Función
	
	{attribute 'OPC.UA.DA' := '1'} 
	Belt_Conveyor_2m_19 AT %Q* : BOOL;
	{attribute 'OPC.UA.DA' := '1'} 
	Belt_Conveyor_2m_20 AT %Q* : BOOL;
	{attribute 'OPC.UA.DA' := '1'} 
	Belt_Conveyor_2m_21 AT %Q* : BOOL;
	{attribute 'OPC.UA.DA' := '1'} 
	Belt_Conveyor_4m_12 AT %Q* : BOOL;
	{attribute 'OPC.UA.DA' := '1'} 
	Belt_Conveyor_4m_13 AT %Q* : BOOL;
	{attribute 'OPC.UA.DA' := '1'} 
	Belt_Conveyor_4m_14 AT %Q* : BOOL;
	{attribute 'OPC.UA.DA' := '1'} 
	Belt_Conveyor_4m_15 AT %Q* : BOOL;
	{attribute 'OPC.UA.DA' := '1'} 
	Belt_Conveyor_Inclined_3 AT %Q* : BOOL;
	//{attribute 'OPC.UA.DA' := '1'}  // Comentar
	Emitter_7 AT %Q* : BOOL := FALSE;
	//{attribute 'OPC.UA.DA' := '1'}  // Comentar
	Palletizer_3_Belt_mas AT %Q* : BOOL;
	//{attribute 'OPC.UA.DA' := '1'}  // Comentar
	Palletizer_3_Chain_mas AT %Q* : BOOL;	
	//{attribute 'OPC.UA.DA' := '1'}  // Comentar
	Palletizer_3_Clamb AT %Q* : BOOL;
	//{attribute 'OPC.UA.DA' := '1'}  // Comentar
	Palletizer_3_Elevator_mas AT %Q* : BOOL;
	//{attribute 'OPC.UA.DA' := '1'}  // Comentar
	Palletizer_3_Elevator_menos AT %Q* : BOOL;
	//{attribute 'OPC.UA.DA' := '1'}  // Comentar
	Palletizer_3_Elevator_Move_Limit AT %Q* : BOOL;
	//{attribute 'OPC.UA.DA' := '1'}  // Comentar
	Palletizer_3_Open_Plate AT %Q* : BOOL;
	//{attribute 'OPC.UA.DA' := '1'}  // Comentar
	Palletizer_3_Push AT %Q* : BOOL;
	//{attribute 'OPC.UA.DA' := '1'}  // Comentar
	Palletizer_3_Turn AT %Q* : BOOL;
	{attribute 'OPC.UA.DA' := '1'} 
	Pivot_Arm_Sorter_4_Turn AT %Q* : BOOL;
	//{attribute 'OPC.UA.DA' := '1'}  // Comentar
	RFID_Reader_3_Ejecute_Comm AT %Q* : BOOL;
	//{attribute 'OPC.UA.DA' := '1'}  // Comentar /
	Right_Positioner_5_Clamp AT %Q* : BOOL;
	//{attribute 'OPC.UA.DA' := '1'}  // Comentar
	Right_Positioner_6_Clamp AT %Q* : BOOL;	
	//{attribute 'OPC.UA.DA' := '1'}  // Comentar
	Right_Positioner_6_Raise AT %Q* : BOOL;	
	{attribute 'OPC.UA.DA' := '1'} 
	Roller_Conveyor_2m_7 AT %Q* : BOOL;
	//{attribute 'OPC.UA.DA' := '1'}  // Comentar
	Two_Axis_Pick_Place_3_Grab AT %Q* : BOOL;
	//{attribute 'OPC.UA.DA' := '1'}  // Comentar
	Two_Axis_Pick_Place_3Z AT %Q* : BOOL;
	//{attribute 'OPC.UA.DA' := '1'}  // Comentar
	Two_Axis_Pick_Place_3X AT %Q* : BOOL;
	
	
//Almacén
	
	{attribute 'OPC.UA.DA' := '1'} 
	Chain_Transfer_1_mas AT %Q* : BOOL;
	{attribute 'OPC.UA.DA' := '1'} 
	Curved_Roller_Conveyor_1_CCW AT %Q* : BOOL;
	{attribute 'OPC.UA.DA' := '1'} 
	Curved_Roller_Conveyor_2_CW AT %Q* : BOOL;
	{attribute 'OPC.UA.DA' := '1'} 
	Digital_Display_1 AT %Q* : DINT;		
	{attribute 'OPC.UA.DA' := '1'} 
	Light_Indicator_Green AT %Q* : BOOL;
	{attribute 'OPC.UA.DA' := '1'} 
	Light_Indicator_Blue AT %Q* : BOOL;
	{attribute 'OPC.UA.DA' := '1'} 
	Light_Indicator_Red	 AT %Q* : BOOL;	
	{attribute 'OPC.UA.DA' := '1'} 
	Loading_Conveyor_1 AT %Q* : BOOL;
	{attribute 'OPC.UA.DA' := '1'} 
	Loading_Conveyor_2 AT %Q* : BOOL;
	//{attribute 'OPC.UA.DA' := '1'} 
	Reset_Button_1_Light AT %Q* : BOOL;
	//{attribute 'OPC.UA.DA' := '1'} 
	Reset_Button_9_Light AT %Q* : BOOL;
	{attribute 'OPC.UA.DA' := '1'} 
	RFID_Reader_4_Command AT %Q* : DINT := 2;
	{attribute 'OPC.UA.DA' := '1'} 
	RFID_Reader_4_Ejecute_Comm AT %Q* : BOOL;
	{attribute 'OPC.UA.DA' := '1'} 
	Roller_Conveyor_2m_2 AT %Q* : BOOL;
	{attribute 'OPC.UA.DA' := '1'} 
	Roller_Conveyor_2m_3 AT %Q* : BOOL;	
	{attribute 'OPC.UA.DA' := '1'} 
	Roller_Conveyor_2m_5 AT %Q* : BOOL;
	{attribute 'OPC.UA.DA' := '1'} 
	Roller_Conveyor_2m_6 AT %Q* : BOOL;	
	{attribute 'OPC.UA.DA' := '1'} 
	Roller_Conveyor_2m_8 AT %Q* : BOOL;
	{attribute 'OPC.UA.DA' := '1'} 
	Roller_Conveyor_2m_9 AT %Q* : BOOL;
	{attribute 'OPC.UA.DA' := '1'} 
	Roller_Conveyor_4m_1 AT %Q* : BOOL;	
	{attribute 'OPC.UA.DA' := '1'} 
	Roller_Conveyor_4m_2 AT %Q* : BOOL;	
	{attribute 'OPC.UA.DA' := '1'} 
	Roller_Conveyor_4m_3 AT %Q* : BOOL;
	{attribute 'OPC.UA.DA' := '1'} 
	Roller_Conveyor_6m_1 AT %Q* : BOOL;
	{attribute 'OPC.UA.DA' := '1'} 
	Roller_Conveyor_6m_2 AT %Q* : BOOL;
	//{attribute 'OPC.UA.DA' := '1'} // Comentar
	Stack_Light_13_Green AT %Q* : BOOL;
	//{attribute 'OPC.UA.DA' := '1'} // Comentar
	Stack_Light_14_Green AT %Q* : BOOL;
	//{attribute 'OPC.UA.DA' := '1'} // Comentar
	Stack_Light_13_Red AT %Q* : BOOL;	
	//{attribute 'OPC.UA.DA' := '1'} // Comentar
	Stack_Light_14_Red AT %Q* : BOOL;	
	//{attribute 'OPC.UA.DA' := '1'} // Comentar
	Stack_Light_13_Yellow AT %Q* : BOOL;		
	//{attribute 'OPC.UA.DA' := '1'} // Comentar
	Stack_Light_14_Yellow AT %Q* : BOOL;
	{attribute 'OPC.UA.DA' := '1'} 
	Stacker_Crane_1_Left AT %Q* : BOOL;
	{attribute 'OPC.UA.DA' := '1'} 
	Stacker_Crane_1_Lift AT %Q* : BOOL;
	{attribute 'OPC.UA.DA' := '1'} 
	Stacker_Crane_1_Right AT %Q* : BOOL;
	{attribute 'OPC.UA.DA' := '1'} 
	Stacker_Crane_1_Target_Position  AT %Q* : DINT;	
	//{attribute 'OPC.UA.DA' := '1'} 
	Start_Button_1_Light AT %Q* : BOOL;
	//{attribute 'OPC.UA.DA' := '1'} 
	Start_Button_9_Light AT %Q* : BOOL;
	//{attribute 'OPC.UA.DA' := '1'} 
	Stop_Button_1_Light AT %Q* : BOOL;
	//{attribute 'OPC.UA.DA' := '1'} 
	Stop_Button_9_Light AT %Q* : BOOL;
	{attribute 'OPC.UA.DA' := '1'} 
	Turnable_1_Turn AT %Q* : BOOL;
	{attribute 'OPC.UA.DA' := '1'} 
	Turnable_1_Roll_menos AT %Q* : BOOL;
	{attribute 'OPC.UA.DA' := '1'} 
	Turnable_2_Turn AT %Q* : BOOL;
	{attribute 'OPC.UA.DA' := '1'} 
	Turnable_2_Roll_menos AT %Q* : BOOL;
	

//Exclusivo HMI
	
	//{attribute 'OPC.UA.DA' := '1'}
	Palletizer_1_Belt_menos AT %Q* : BOOL;
	//{attribute 'OPC.UA.DA' := '1'} 
	Palletizer_1_Chain_menos AT %Q* : BOOL;	
	//{attribute 'OPC.UA.DA' := '1'}  
	Two_Axis_Pick_Place_1_Gripper_CCW AT %Q* : BOOL;	
	//{attribute 'OPC.UA.DA' := '1'}  
	Two_Axis_Pick_Place_1_Gripper_CW AT %Q* : BOOL;
	//{attribute 'OPC.UA.DA' := '1'} 
	Two_Axis_Pick_Place_1_Rotate_CCW AT %Q* : BOOL := FALSE;	
	//{attribute 'OPC.UA.DA' := '1'} 
	Two_Axis_Pick_Place_1_Rotare_CW AT %Q* : BOOL := FALSE;
	//{attribute 'OPC.UA.DA' := '1'}
	Palletizer_2_Belt_menos AT %Q* : BOOL;	
	//{attribute 'OPC.UA.DA' := '1'}
	Palletizer_2_Chain_menos AT %Q* : BOOL;	
	//{attribute 'OPC.UA.DA' := '1'}  
	Two_Axis_Pick_Place_2_Gripper_CCW AT %Q* : BOOL;	
	//{attribute 'OPC.UA.DA' := '1'}  
	Two_Axis_Pick_Place_2_Gripper_CW AT %Q* : BOOL;
	//{attribute 'OPC.UA.DA' := '1'} 
	Two_Axis_Pick_Place_2_Rotate_CCW AT %Q* : BOOL := FALSE;	
	//{attribute 'OPC.UA.DA' := '1'} 
	Two_Axis_Pick_Place_2_Rotare_CW AT %Q* : BOOL := FALSE;	
	//{attribute 'OPC.UA.DA' := '1'}
	Palletizer_3_Belt_menos AT %Q* : BOOL;	
	//{attribute 'OPC.UA.DA' := '1'}
	Palletizer_3_Chain_menos AT %Q* : BOOL;	
	//{attribute 'OPC.UA.DA' := '1'} 
	Pivot_Arm_Sorter_1_Turn AT %Q* : BOOL;	
	//{attribute 'OPC.UA.DA' := '1'} 
	Pivot_Arm_Sorter_2_Belt_menos AT %Q* : BOOL;
	//{attribute 'OPC.UA.DA' := '1'} 
	Pivot_Arm_Sorter_3_Belt_menos AT %Q* : BOOL;
	//{attribute 'OPC.UA.DA' := '1'} 
	Pivot_Arm_Sorter_4_Belt_menos AT %Q* : BOOL;
	//{attribute 'OPC.UA.DA' := '1'}  
	RFID_Reader_1_Memory_Index AT %Q* : DINT;
	//{attribute 'OPC.UA.DA' := '1'}  
	RFID_Reader_2_Memory_Index AT %Q* : DINT;
	//{attribute 'OPC.UA.DA' := '1'}  
	RFID_Reader_3_Memory_Index AT %Q* : DINT;
	//{attribute 'OPC.UA.DA' := '1'}  
	RFID_Reader_4_Memory_Index AT %Q* : DINT;
	//{attribute 'OPC.UA.DA' := '1'} 
	Right_Positioner_1_Raise AT %Q* : BOOL;	
	//{attribute 'OPC.UA.DA' := '1'} 
	Right_Positioner_3_Raise AT %Q* : BOOL;		
	//{attribute 'OPC.UA.DA' := '1'} 
	Right_Positioner_5_Raise AT %Q* : BOOL;	
	//{attribute 'OPC.UA.DA' := '1'} 
	Turnable_1_Roll_mas AT %Q* : BOOL;
	//{attribute 'OPC.UA.DA' := '1'} 
	Turnable_2_Roll_mas AT %Q* : BOOL;	
	//{attribute 'OPC.UA.DA' := '1'}  
	Two_Axis_Pick_Place_3_Gripper_CCW AT %Q* : BOOL;	
	//{attribute 'OPC.UA.DA' := '1'}  
	Two_Axis_Pick_Place_3_Gripper_CW AT %Q* : BOOL;
	//{attribute 'OPC.UA.DA' := '1'} 
	Two_Axis_Pick_Place_3_Rotate_CCW AT %Q* : BOOL := FALSE;	
	//{attribute 'OPC.UA.DA' := '1'} 
	Two_Axis_Pick_Place_3_Rotare_CW AT %Q* : BOOL := FALSE;

	
	
END_VAR

// ---- POUs/Almacén/FUN_get_Posicion_Ocupada_Array.TcPOU
FUNCTION FUN_get_Posicion_Ocupada_Array : INT
VAR_INPUT
	color : INT;
END_VAR
VAR
	i 				: INT;
	ContadorPalets 	: INT  := 0;
	ocupada 		: BOOL := TRUE;	
END_VAR


// Retorna la primera posicion ocupada del color correspondiente en el array Clasificados
FOR i := 0 TO 53 DO
	IF GVL.Clasificados[i].Color = color THEN
		ContadorPalets := ContadorPalets +1;
		IF ocupada THEN
			FUN_get_Posicion_Ocupada_Array := i+1;
			ocupada := FALSE;
		END_IF
	END_IF
END_FOR

IF ocupada THEN
	FUN_get_Posicion_Ocupada_Array := 0;
END_IF

GVL.ContadorPalets := ContadorPalets;

END_FUNCTION

// ---- POUs/Almacén/POU_Almacen.TcPOU
PROGRAM POU_Almacen
VAR
	
	bGetTime    				: BOOL; // Trigger para obtener el tiempo
	Color						: DINT 	:= 0; // Color del producto del palet a almacenar
	Color_Retirada				: INT  	:= 0; // Color del producto del palet a retirar del Almacen
	fbLocalTime 				: FB_LocalSystemTime := ( bEnable := TRUE, sNetID := '10.24.136.19.1.1',dwcycle := 100);
	Hay_Palet 					: BOOL	:= FALSE; // variable para indicar si hay un palet en posición para ser recogido pro la grúa
	MovingZ						: BOOL 	:= FALSE; // Variable de control que indica si la grúa ha dejado de moverse en el eje Z
	MovingX						: BOOL 	:= FALSE; // Variable de control que indica si la grúa ha dejado de moverse en el eje X	
	Pallet_Almacen_I 			: CTUD; // Contador de palet en la última cinta antes del almacén
	posicion					: INT; // posición del palet a almacenar/retirar
	posLibre					: INT; // primera posición libre del almacen
	Posicion_Extraer_Antigua	: INT  	:= 0; // Posicion del palet a extraer en el almacen
	FB_Visibilidad 				: FB_Visibilidad;
END_VAR

 // ---------------------------------------------------------------- 1. FALLING Y RASING EDGES ----------------------------------------------------------------

IF POU_Edges.FallingEdgeZ.Q THEN
	MovingZ := TRUE;
END_IF

IF POU_Edges.FallingEdgeX.Q THEN
	MovingX := TRUE;
END_IF


IF POU_Edges.Falling_Edge_Almacen_I_R.Q THEN Hay_Palet := TRUE; END_IF // Cuando llega el palet al final del loading, se indica que está lista para ser almacenada

 // ---------------------------------------------------------------- 2. CONTROL CINTAS ----------------------------------------------------------------
 
Pallet_Almacen_I (CU:= POU_Edges.Rasing_Edge_Almacen_I_D.Q,CD := POU_Edges.Falling_Edge_Almacen_I_2.Q);

GVL.Loading_Conveyor_1 := (NOT Hay_Palet AND WORD_TO_INT(Pallet_Almacen_I.CV) =1); // Si el palet no está posicionado para ser guardado(ha llegado al final) pero se está posicionando
GVL.Roller_Conveyor_2m_8 := NOT (GVL.Diffuse_Sensor_43 AND  WORD_TO_INT(Pallet_Almacen_I.CV) >1) AND GVL.Contador_Linea_Cruce_2>0;	// Si hay un palet en el Loading y aparece otro, se para la cinta

 // ---------------------------------------------------------------- 3. MODO ALMACENAMIENTO ----------------------------------------------------------------

IF GVL.Control_Almacen THEN	
	CASE GVL.Estado_Almacen_I OF
		
		0: //Estado 0, leemos la información del palet
			IF Hay_Palet THEN
				GVL.RFID_Reader_4_Ejecute_Comm := TRUE;
				GVL.Estado_Almacen_I := 1;
			END_IF
		
		1: 	//Estado 1, le damos un estado de espera para comprobar si ha escrito bien
			IF GVL.RFID_Reader_4_Status=0 AND GVL.Pallets_Almacenados = GVL.RFID_Reader_4_Command_ID THEN			
				RFID_Reader_4_Ejecute_Comm := FALSE;			
				Color := GVL.RFID_Reader_4_Read_Data;
				
				IF	GVL.RFID_Reader_4_Status=0 THEN
					GVL.Error_RFID_Almacen := FALSE;
				ELSE						
					GVL.Error_RFID_Almacen := TRUE;	
				END_IF
				
				GVL.Estado_Almacen_I := 2;
				
			END_IF
			
		2: // Estado 2, extendemos para coger palet
			posLibre := FUN_get_Posicion_Libre_Array();
			IF  NOT GVL.Retroreflective_Sensor_1 AND posLibre <> 0 AND NOT GVL.Retirada_Start AND Estado_Almacen_O =1THEN
				GVL.Stacker_Crane_1_Right := TRUE;
				GVL.Estado_Almacen_I := 3;
			END_IF
		
		3: // Estado 3, levantamos para coger la palet 
			IF  GVL.Stacker_Crane_1_Right_Limit  THEN
				GVL.Stacker_Crane_1_Lift := TRUE;
				GVL.Estado_Almacen_I := 4;
			END_IF
			
		4: // Estado 4, una vez levantada, volvemos
			IF  POU_Edges.FallingEdgeZ.Q THEN
				GVL.Stacker_Crane_1_Right := FALSE;				
				Hay_Palet := FALSE;
			END_IF
			
		5: // Estado 5, llevamos a guardarla
			IF GVL.Stacker_Crane_1_Middle_Limit THEN	
				
				IF GVL.Error_RFID_Almacen THEN	
					GVL.Stacker_Crane_1_Left := TRUE;
					GVL.Estado_Almacen_I := 7 ;	
				ELSE
					MovingZ  := FALSE;
					posicion := FUN_get_Posicion_Libre_Array();
					GVL.Stacker_Crane_1_Target_Position:= posicion; // recorremos el array hasta obtener la primera posición a guardar
					GVL.Clasificados[posicion-1].Color := Color;	
					FB_Visibilidad(Color:= Color, Posicion:= Posicion);
					IF fbLocalTime.bValid THEN   				 
						GVL.Clasificados[posicion-1].Fecha_Hora := SYSTEMTIME_TO_DT(fbLocalTime.systemTime);
					END_IF;
					GVL.Estado_Almacen_I := 6;
				END_IF
				
			END_IF
			
		6: // Estado 6, llegados a la posición expandimos para colocar el palet
			IF MovingX AND MovingZ THEN
				GVL.Stacker_Crane_1_Left := TRUE;
				MovingX  := FALSE;
				MovingZ  := FALSE;
				GVL.Estado_Almacen_I := 7;
			END_IF
			
		7: //Estado 7, una vez expandida bajamos para dejarla posicionada
			IF GVL.Stacker_Crane_1_Left_Limit  THEN
				// Rellenamos el tipo de palet que hay en la posicion	
				GVL.Stacker_Crane_1_Lift := FALSE;
				GVL.Estado_Almacen_I := 8;	
				
			END_IF
			
		8: // Estado 8, una vez bajada recojemos
			IF MovingZ  THEN
				// Rellenamos el tipo de palet que hay en la posicion
				GVL.Stacker_Crane_1_Left := FALSE;
				MovingZ  := FALSE;
				GVL.Estado_Almacen_I := 9;
			END_IF
		
		9: // Estado 9, volvemos a reposo
			IF GVL.Stacker_Crane_1_Middle_Limit THEN
				
				IF GVL.Error_RFID_Almacen THEN					
					GVL.Estado_Almacen_I := 0;
				ELSE
					GVL.Stacker_Crane_1_Target_Position := 55 ;
					GVL.Estado_Almacen_I :=10;
				END_IF
				
			END_IF
			
		10: // Estado 10, esperamos hasta que llegue a la posición de reposo
			IF MovingZ AND MovingX THEN
				GVL.Roller_Conveyor_2m_1 := TRUE;
				GVL.Loading_Conveyor_1 :=TRUE;
				MovingX  := FALSE;
				MovingZ  := FALSE;
				GVL.Estado_Almacen_I := 0;
			END_IF
			
	END_CASE
END_IF

 // ---------------------------------------------------------------- 3. MODO EXTRACCIÓN ----------------------------------------------------------------

// FUNCIONES SELECTOR (1: Azul, 4:Verde, 7:Metal)

IF GVL.Selector1_State_1 THEN 
	
	Color_Retirada := 4;
	GVL.Light_Indicator_Green := TRUE;
	GVL.Light_Indicator_Blue := FALSE;
	GVL.Light_Indicator_Red := FALSE;

// Extraer Metal
ELSIF GVL.Selector1_State_2 THEN 
	
	Color_Retirada := 7;
	GVL.Light_Indicator_Green := FALSE;
	GVL.Light_Indicator_Blue := FALSE;
	GVL.Light_Indicator_Red := TRUE;
	
// Extraer Azul	
ELSE 
	
	Color_Retirada := 1;
	GVL.Light_Indicator_Green := FALSE;
	GVL.Light_Indicator_Blue := TRUE;
	GVL.Light_Indicator_Red := FALSE;
	
END_IF

posicion := FUN_get_Posicion_Ocupada_Array(Color_Retirada);
GVL.Digital_Display_1 := GVL.ContadorPalets;


// MOVIMIENTOS DE LA GRÚA

IF GVL.Control_Almacen THEN	
	CASE GVL.Estado_Almacen_O OF
	
		1: // Estado 1, Si se ha pulsado el boton de Start y hay Palets a retirar del material seleccionado, enviamos la grua a recoger el palet
			IF GVL.Retirada_Start  AND Estado_Almacen_I =2 AND posicion<>0 THEN	
				GVL.Stacker_Crane_1_Target_Position:= posicion; // Se recorre el array para obtener la primera posición libre
				Posicion_Extraer_Antigua := posicion;
				GVL.Estado_Almacen_O := 2;
			END_IF
			
		2: // Estado 2, llegados a la posición expandimos para recoger el palet
			IF MovingX AND MovingZ THEN
				GVL.Stacker_Crane_1_Left := TRUE;
				MovingX  := FALSE;
				MovingZ  := FALSE;
				GVL.Estado_Almacen_O := 3;
			END_IF
				
		3: //Estado 3, una vez expandida subirmos para recoger el palet
			IF GVL.Stacker_Crane_1_Left_Limit THEN
				GVL.Stacker_Crane_1_Lift := TRUE;
				GVL.Estado_Almacen_O := 4;				
			END_IF
	
			
		4: // Estado 4, una vez subida recojemos y liberamos al posición del array
			IF MovingZ THEN
				GVL.Stacker_Crane_1_Left := FALSE;
				MovingZ  := FALSE;;
				GVL.Clasificados[Posicion_Extraer_Antigua-1].Color := 0;
				GVL.Clasificados[Posicion_Extraer_Antigua-1].Fecha_Hora := DT#1999-01-01-00:00:00;				
				FB_Visibilidad(Color:= 0, Posicion:= Posicion_Extraer_Antigua);
				GVL.Estado_Almacen_O := 5;	
			END_IF
			
		5: // Estado 5, volvemos a reposo
			IF GVL.Stacker_Crane_1_Middle_Limit THEN
				GVL.Stacker_Crane_1_Target_Position := 55 ;
				GVL.Estado_Almacen_O := 6;
			END_IF
			
		6: // Estado 6, extendemos para colocar palet
			IF  MovingX AND MovingZ THEN
				GVL.Loading_Conveyor_2 :=FALSE;
				GVL.Stacker_Crane_1_Left := TRUE;
				MovingX  := FALSE;
				MovingZ  := FALSE;
				GVL.Estado_Almacen_O := 7 ;
			END_IF
			
		7: // Estado 7, bajamos para soltar la palet 
			IF  GVL.Stacker_Crane_1_Left_Limit THEN
				GVL.Stacker_Crane_1_Lift := FALSE;
				GVL.Estado_Almacen_O := 8;
			END_IF
			
		8: // Estado 8, una vez bajada, volvemos
			IF  MovingZ THEN
				GVL.Stacker_Crane_1_Left := FALSE;
				GVL.Estado_Almacen_O := 9;
				MovingZ  := FALSE;
				//GVL.Loading_Conveyor_2 := TRUE;
			END_IF
			
		9: // Estado 9, esperamos hasta que llegue a la posición de reposo
			IF GVL.Stacker_Crane_1_Middle_Limit THEN
				GVL.Estado_Almacen_O := 1;
			END_IF
	
	END_CASE
END_IF

END_PROGRAM

// ---- POUs/Control funcionalidad/POU_Edges.TcPOU
PROGRAM POU_Edges
VAR
		
	// Falling Edges
	
	Falling_Edge_Almacen_I_2 			: F_TRIG;
	Falling_Edge_Almacen_I_D 			: F_TRIG;
	Falling_Edge_Almacen_I_R			: F_TRIG;
	Falling_Edge_Almacen_O 				: F_TRIG;
	Falling_Edge_Azul_Separada 			: F_TRIG;
	Falling_Edge_Cruce_1_F 				: F_TRIG;
	Falling_Edge_Cruce_1_I 				: F_TRIG;
	Falling_Edge_Cruce_1_Salida 		: F_TRIG;
	Falling_Edge_Cruce_2_F 				: F_TRIG;	
	Falling_Edge_Cruce_2_I 				: F_TRIG;
	Falling_Edge_Cruce_2_Salida 		: F_TRIG;	
	Falling_Edge_Descartadas 			: F_TRIG;
	Falling_Edge_Diff_6 				: F_TRIG;
	Falling_Edge_Diff_7 				: F_TRIG;
	Falling_Edge_Diff_10 				: F_TRIG;
	Falling_Edge_Diff_11 				: F_TRIG;
	Falling_Edge_Diff_13 				: F_TRIG;
	Falling_Edge_Diff_14 				: F_TRIG;
	Falling_Edge_Entrada_Manipulador_1 	: F_TRIG;
	Falling_Edge_Entrada_Manipulador_2 	: F_TRIG;
	Falling_Edge_Entrada_Manipulador_3 	: F_TRIG;
	Falling_Edge_Entrada_Manipulador_4 	: F_TRIG;
	Falling_Edge_Entrada_Manipulador_5 	: F_TRIG;
	Falling_Edge_Entrada_Manipulador_6 	: F_TRIG;	
	Falling_Edge_Limpiador 				: F_TRIG; 
	Falling_Edge_Metal_Separada 		: F_TRIG;
	Falling_Edge_Paletizador_1 			: F_TRIG; 
	Falling_Edge_Paletizador_2 			: F_TRIG;
	Falling_Edge_Paletizador_3 			: F_TRIG;
	Falling_Edge_Sensor_Salida_C1 		: F_TRIG;
	Falling_Edge_Sensor_Salida_C2 		: F_TRIG;
	Falling_Edge_Sensor_Secundario_C1 	: F_TRIG;
	Falling_Edge_Sensor_Secundario_C2 	: F_TRIG;
	Falling_Edge_Sensor_Zona_Azul 		: F_TRIG;
	Falling_Edge_Sensor_Zona_Metal 		: F_TRIG;
	Falling_Edge_Sensor_Zona_Verde 		: F_TRIG;
	Falling_Edge_Verde_Separada 		: F_TRIG;
	FallingEdgeZ						: F_TRIG;
	FallingEdgeX						: F_TRIG;
	
	// Rasing Edges
	
	Rasing_Edge_Almacen_I_D 			: R_TRIG;
	Rasing_Edge_Almacen_O 				: R_TRIG;
	Rasing_Edge_Diff_6 					: R_TRIG;
	Rasing_Edge_Diff_7 					: R_TRIG;
	Rasing_Edge_Diff_10 				: R_TRIG;
	Rasing_Edge_Diff_11 				: R_TRIG;
	Rasing_Edge_Diff_13 				: R_TRIG;
	Rasing_Edge_Diff_14 				: R_TRIG;	
	Rasing_Edge_Emisor 					: R_TRIG;
	Rasing_Edge_Limpiador 				: R_TRIG;
	Rasing_Edge_Salida_Manipulador_1 	: R_TRIG;
	Rasing_Edge_Salida_Manipulador_2 	: R_TRIG;
	Rasing_Edge_Salida_Manipulador_3 	: R_TRIG;
	Rasing_Edge_Salida_Manipulador_4 	: R_TRIG;
	Rasing_Edge_Salida_Manipulador_5 	: R_TRIG;
	Rasing_Edge_Salida_Manipulador_6 	: R_TRIG;	
	Rasing_Edge_Sensor_Principal_C1 	: R_TRIG;
	Rasing_Edge_Sensor_Principal_C2 	: R_TRIG;
	Rasing_Edge_Sensor_Zona_Azul		: R_TRIG;
	
	
END_VAR

//Etapa1
Falling_Edge_Sensor_Zona_Azul(CLK:=GVL.Diffuse_Sensor_2);
Falling_Edge_Sensor_Zona_Metal(CLK:=GVL.Diffuse_Sensor_4);
Falling_Edge_Sensor_Zona_Verde(CLK:=GVL.Diffuse_Sensor_3);
Rasing_Edge_Sensor_Zona_Azul(CLK:=GVL.Diffuse_Sensor_2);

// Linea Principal
Falling_Edge_Azul_Separada(CLK:=GVL.Diffuse_Sensor_5);
Falling_Edge_Descartadas (CLK:= GVL.Diffuse_Sensor_8);
Falling_Edge_Limpiador(CLK:=GVL.Diffuse_Sensor_2);
Rasing_Edge_Emisor(CLK:=GVL.Diffuse_Sensor_0);
Rasing_Edge_Limpiador(CLK:=GVL.Diffuse_Sensor_2);

// Linea Azul
Falling_Edge_Diff_6 (CLK:=GVL.Diffuse_Sensor_6);
Falling_Edge_Diff_7 (CLK:=GVL.Diffuse_Sensor_7);
Falling_Edge_Entrada_Manipulador_1 (CLK:=GVL.Diffuse_Sensor_15);
Falling_Edge_Entrada_Manipulador_2 (CLK:=GVL.Diffuse_Sensor_16);
Falling_Edge_Paletizador_1 (CLK:=GVL.Palletizer_1_Elevator_Front_Limit); 
Rasing_Edge_Diff_6 (CLK:=GVL.Diffuse_Sensor_6);
Rasing_Edge_Diff_7 (CLK:=GVL.Diffuse_Sensor_7);
Rasing_Edge_Salida_Manipulador_1 (CLK:=GVL.Diffuse_Sensor_17);
Rasing_Edge_Salida_Manipulador_2 (CLK:=GVL.Diffuse_Sensor_18);

//Linea Verde
Falling_Edge_Diff_10 (CLK:=GVL.Diffuse_Sensor_10);
Falling_Edge_Diff_11 (CLK:=GVL.Diffuse_Sensor_11);
Falling_Edge_Entrada_Manipulador_3 (CLK:=GVL.Diffuse_Sensor_23);
Falling_Edge_Entrada_Manipulador_4 (CLK:=GVL.Diffuse_Sensor_24);
Falling_Edge_Paletizador_2 (CLK:=GVL.Palletizer_2_Elevator_Front_Limit); 
Rasing_Edge_Diff_10 (CLK:=GVL.Diffuse_Sensor_10);
Rasing_Edge_Diff_11 (CLK:=GVL.Diffuse_Sensor_11);
Rasing_Edge_Salida_Manipulador_3 (CLK:=GVL.Diffuse_Sensor_25);
Rasing_Edge_Salida_Manipulador_4 (CLK:=GVL.Diffuse_Sensor_26);
Falling_Edge_Verde_Separada(CLK:=GVL.Diffuse_Sensor_9);

//Linea Metal
Falling_Edge_Diff_13 (CLK:=GVL.Diffuse_Sensor_13);
Falling_Edge_Diff_14 (CLK:=GVL.Diffuse_Sensor_14);
Falling_Edge_Entrada_Manipulador_5 (CLK:=GVL.Diffuse_Sensor_31);
Falling_Edge_Entrada_Manipulador_6 (CLK:=GVL.Diffuse_Sensor_32);
Falling_Edge_Metal_Separada(CLK:=GVL.Diffuse_Sensor_12);
Falling_Edge_Paletizador_3 (CLK:=GVL.Palletizer_3_Elevator_Front_Limit); 
Rasing_Edge_Diff_14 (CLK:=GVL.Diffuse_Sensor_14);
Rasing_Edge_Diff_13 (CLK:=GVL.Diffuse_Sensor_13);
Rasing_Edge_Salida_Manipulador_5 (CLK:=GVL.Diffuse_Sensor_33);
Rasing_Edge_Salida_Manipulador_6 (CLK:=GVL.Diffuse_Sensor_34);

// Cruce 1
Rasing_Edge_Sensor_Principal_C1 (CLK := GVL.Diffuse_Sensor_39);
Falling_Edge_Sensor_Salida_C1 (CLK := GVL.Turnable_1_Back_Limit);
Falling_Edge_Sensor_Secundario_C1 (CLK := GVL.Diffuse_Sensor_40);

// Cruce 2
Rasing_Edge_Sensor_Principal_C2 (CLK := GVL.Diffuse_Sensor_41);
Falling_Edge_Sensor_Salida_C2 (CLK := GVL.Turnable_2_Back_Limit);
Falling_Edge_Sensor_Secundario_C2 (CLK := GVL.Diffuse_Sensor_42);

//Linea Almacen
Falling_Edge_Cruce_1_I (CLK:=GVL.Diffuse_Sensor_39);
Falling_Edge_Cruce_1_F (CLK:=GVL.Diffuse_Sensor_40);
Falling_Edge_Cruce_2_I (CLK:=GVL.Diffuse_Sensor_41);
Falling_Edge_Cruce_2_f (CLK:=GVL.Diffuse_Sensor_42);
Falling_Edge_Cruce_1_Salida (CLK := GVL.Turnable_1_Back_Limit); 
Falling_Edge_Cruce_2_Salida (CLK := GVL.Turnable_2_Back_Limit);
Falling_Edge_Almacen_I_D (CLK := GVL.Diffuse_Sensor_43);
Falling_Edge_Almacen_O (CLK := GVL.Diffuse_Sensor_44);
Rasing_Edge_Almacen_O (CLK := GVL.Retroreflective_Sensor_2);

// Almacen
FallingEdgeX(CLK:=GVL.Stacker_Crane_1_Moving_X, Q=> );
FallingEdgeZ(CLK:=GVL.Stacker_Crane_1_Moving_Z, Q=> );
Falling_Edge_Almacen_I_R(CLK:=GVL.Retroreflective_Sensor_1, Q=> );
Rasing_Edge_Almacen_I_D (CLK := GVL.Diffuse_Sensor_43);
Falling_Edge_Almacen_I_2 (CLK := POU_Almacen.Hay_Palet);

END_PROGRAM

// ---- POUs/Almacén/POU_Cruce_Almacen.TcPOU
FUNCTION_BLOCK POU_Cruce_Almacen
VAR_INPUT
	
	Contador_Corto 					: INT; // Contador de la palets en la cinta de rodillos corta a la entrada del cruce
	Contador_Largo 					: INT; // Contador de la palets en la cinta de rodillos larga a la entrada del cruce
	Diffuse_Sensor_Corto 			: BOOL; // Sensor en la cinta de rodillos corta a la entrada del cruce
	Diffuse_Sensor_Largo			: BOOL; // Sensor en la cinta de rodillos larga a la entrada del cruce
	Falling_Edge_Sensor_Salida 		: BOOL;
	Falling_Edge_Sensor_Secundario 	: BOOL;
	Rasing_Edge_Sensor_Principal	: BOOL;	
	Sacar_Palet_Paletizador			: BOOL; // Variable para indicar que el paletizador puede introducir el palet ya relleno en la cinta de salida
	Sacar_Palet_Turntable			: BOOL; // Variable para indicar que la plataforma giratoria puede introducir el palet en la cinta principal
	Turnable_Back_Limit 			: BOOL; // Sensor trasero de la plataforma giratoria
	Turnable_Limit_0 				: BOOL; // Sensor de límite 0 de la plataforma giratoria
	Turnable_Limit_90 				: BOOL; // Sensor de límite 90 de la plataforma giratoria
	
END_VAR
VAR_OUTPUT
	
	Roller_Conveyor_Corto 			: BOOL; // Cinta transportadora de la línea corta de entrada
	Roller_Conveyor_Largo 			: BOOL; // Cinta transportadora de la línea larga de entrada
	Turnable_Roll_menos 			: BOOL := FALSE; // Variable relacionada con los rodillos de la plataforma giratoria
	Turnable_Turn 					: BOOL := TRUE; // Variable relacionada con el giro de la plataforma
	
END_VAR
VAR
	palet : INT := 0;
END_VAR


//Selección estado del cruce. Si llegan las dos Palets a la vez se le da prioridad a la linea corta, parando la larga	
IF Diffuse_Sensor_Largo AND Diffuse_Sensor_Corto AND palet = 0 THEN // Si no hay palet siendo posicionado y llegan palets a la vez, se posicionará la que haya en la cinta corta
	palet := 2;
ELSIF Diffuse_Sensor_Largo AND palet = 0 THEN // Si no hay palet siendo posicionado y llega una por la línea larga se posicionará
	palet := 1;
ELSIF Diffuse_Sensor_Corto AND palet = 0 THEN // Si no hay palet siendo posicionado y llega una por la línea corta se posicionará
	palet := 2;
END_IF

// Se indica que no hay palet cuando este sale del turntable
IF Falling_Edge_Sensor_Salida THEN
	palet := 0;
END_IF

// Control cintas. Se dejará pasar el palet siempre y cuando la línea de salida esté libre
CASE palet OF
	
	0: // Si no hay palets siendo posicionados, pero hay palets en las líneas para ser posicionadas, muevo las cintas para que lleguen	
		Turnable_Turn := Contador_Largo>0;
		Roller_Conveyor_Largo := Contador_Largo>0;
		Roller_Conveyor_Corto := Sacar_Palet_Paletizador OR (Contador_Corto>0 AND Contador_Corto<2);	
		Turnable_Roll_menos := FALSE;
		
	1: // Accion para trasladar el palet de la izquierda
		Turnable_Turn := TRUE;
		Turnable_Roll_menos := Turnable_Limit_90 AND Sacar_Palet_Turntable;	// Si está en posición y la linea de salida está libre	
		Roller_Conveyor_Largo := (Turnable_Limit_90 AND (NOT Turnable_Back_Limit OR NOT Diffuse_Sensor_Largo)) AND Sacar_Palet_Turntable; // Si está en posición, la línea de salida está libre y no hay palet siendo posicionado		
		Roller_Conveyor_Corto := NOT Diffuse_Sensor_Corto AND (Sacar_Palet_Paletizador OR (Contador_Corto>0 AND Contador_Corto<2)); // Si no hay palet en la línea y el paletizado quiere introducir una
		
	2: // Accion para posicionar el palet de enfrente
		Turnable_Turn := FALSE;		
		Turnable_Roll_menos := Turnable_Limit_0 AND NOT Turnable_Back_Limit; // Se mueve si está en posición y el palet no ha llegado al final
		Roller_Conveyor_Largo := NOT Diffuse_Sensor_Largo; // Si hay un palet, se para la cinta
		// Si está en posición y no acaba de llegar un palet(es decir, o no hay o hay uno en posición) y en la cinta hay un palet o se quiere introducir uno
		Roller_Conveyor_Corto := (Turnable_Limit_0 AND NOT Falling_Edge_Sensor_Secundario)AND (Sacar_Palet_Paletizador OR (Contador_Corto>0 AND Contador_Corto<2)); 
		IF Turnable_Back_Limit THEN // Si viene de colocar la de enfrente y está en el centro, se pasa al estado 3
			palet :=3;
		END_IF		
		
	3: // Accion para trasladar el palet de enfrente ya posicionado
		Turnable_Turn := TRUE;
		Turnable_Roll_menos := Turnable_Limit_90 AND Sacar_Palet_Turntable; // Si está en posición y la línea de enfrente está libre
		Roller_Conveyor_Largo := NOT Diffuse_Sensor_Largo; // Si hay un palet, se para la cinta
		Roller_Conveyor_Corto := NOT Diffuse_Sensor_Corto AND (Sacar_Palet_Paletizador OR (Contador_Corto>0 AND Contador_Corto<2));	// Si no hay palet en la línea y el paletizado quiere introducir una

		
END_CASE

END_FUNCTION_BLOCK

// ---- POUs/Almacén/POU_Linea_Almacen.TcPOU
PROGRAM POU_Linea_Almacen
VAR

	Cruce_1 : POU_Cruce_Almacen;
	Cruce_2 : POU_Cruce_Almacen;
	
END_VAR

// ---------------------------------------------------------------- 1. CRUCES ----------------------------------------------------------------

Cruce_1 (
	Contador_Corto :=GVL.Contador_Palets_Verdes,
	Contador_Largo :=GVL.Contador_Palets_Azules,
	Diffuse_Sensor_Corto := GVL.Diffuse_Sensor_40,
	Diffuse_Sensor_Largo:= GVL.Diffuse_Sensor_39,
	Falling_Edge_Sensor_Salida :=POU_Edges.Falling_Edge_Sensor_Salida_C1.Q,
	Falling_Edge_Sensor_Secundario :=POU_Edges.Falling_Edge_Sensor_Secundario_C1.Q,
	Rasing_Edge_Sensor_Principal :=POU_Edges.Rasing_Edge_Sensor_Principal_C1.Q,
	Sacar_Palet_Paletizador := GVL.Sacar_Palet_2,
	Sacar_Palet_Turntable := GVL.Contador_Linea_Cruce_1 <5,
	Turnable_Back_Limit := GVL.Turnable_1_Back_Limit,	
	Turnable_Limit_0 :=GVL.Turnable_1_Limit_0,
	Turnable_Limit_90 :=GVL.Turnable_1_Limit_90,
	Roller_Conveyor_Corto => GVL.Roller_Conveyor_2m_4 ,
	Roller_Conveyor_Largo => GVL.Roller_Conveyor_4m_1,
	Turnable_Roll_menos => GVL.Turnable_1_Roll_menos,
	Turnable_Turn => GVL.Turnable_1_Turn );
	
Cruce_2 (
	Contador_Corto :=GVL.Contador_Palets_Metal,
	Contador_Largo :=GVL.Contador_Linea_Cruce_2,
	Diffuse_Sensor_Corto := GVL.Diffuse_Sensor_42,
	Diffuse_Sensor_Largo:= GVL.Diffuse_Sensor_41,
	Falling_Edge_Sensor_Salida :=POU_Edges.Falling_Edge_Sensor_Salida_C2.Q,
	Falling_Edge_Sensor_Secundario :=POU_Edges.Falling_Edge_Sensor_Secundario_C2.Q,
	Rasing_Edge_Sensor_Principal :=POU_Edges.Rasing_Edge_Sensor_Principal_C2.Q,
	Sacar_Palet_Paletizador := GVL.Sacar_Palet_3,
	Sacar_Palet_Turntable := GVL.Contador_Linea_Cruce_2 <3,
	Turnable_Back_Limit := GVL.Turnable_2_Back_Limit,	
	Turnable_Limit_0 :=GVL.Turnable_2_Limit_0,
	Turnable_Limit_90 :=GVL.Turnable_2_Limit_90,
	Roller_Conveyor_Corto => GVL.Roller_Conveyor_2m_7 ,
	Roller_Conveyor_Largo => GVL.Roller_Conveyor_2m_5,
	Turnable_Roll_menos => GVL.Turnable_2_Roll_menos,
	Turnable_Turn => GVL.Turnable_2_Turn );
	

// ---------------------------------------------------------------- 2. ALMACEN ----------------------------------------------------------------

POU_Almacen();

END_PROGRAM

// ---- POUs/Control funcionalidad/Contadores_Control_Lineas.TcPOU
PROGRAM Contadores_Control_Lineas
VAR
	// Sumadores
	Contador_Azul 						: CTU;
	Contador_Palets_Azules_Totales 		: CTU;
	Contador_Palets_Metales_Totales 	: CTU;
	Contador_Palets_Verdes_Totales 		: CTU;
	Contador_Emisor						: CTU;
	Contador_Metal						: CTU;
	Contador_Piezas_Descartadas_Totales	: CTU;
	Contador_Verde						: CTU;
	Pallets_Almacenados 				: CTU;
	Pallets_Almacenados_Retirados 		: CTU;
	
	// Sumador-restador
	
	Contador_Palets_Azules 				: CTUD;
	Contador_Palets_Verdes				: CTUD;
	Contador_Linea_Cruce_1 				: CTUD;
	Contador_Linea_Cruce_2 				: CTUD;	
	Contador_Linea_Manipulador_1_I		: CTUD;
	Contador_Linea_Manipulador_2_I		: CTUD;
	Contador_Linea_Manipulador_3_I		: CTUD;
	Contador_Linea_Manipulador_4_I		: CTUD;
	Contador_Linea_Manipulador_5_I		: CTUD;
	Contador_Linea_Manipulador_6_I		: CTUD;
	Contador_Linea_Principal			: CTUD;
	Contador_Manipulador_1				: CTUD;
	Contador_Manipulador_2				: CTUD;
	Contador_Manipulador_3				: CTUD;
	Contador_Manipulador_4				: CTUD;
	Contador_Manipulador_5				: CTUD;
	Contador_Manipulador_6				: CTUD;
	Contador_No_Descartadas				: CTUD;
	Contador_Pivot_Azul					: CTUD;	
	Contador_Pivot_Metal				: CTUD;
	Contador_Pivot_Verde				: CTUD;
	Contador_Zona_Pivot					: CTUD;	
	Pallet_Almacen_O 					: CTUD;
	
	
	
	
END_VAR

// ---------------------------------------------------------------- CONTADORES ----------------------------------------------------------------

//LINEA PRINCIPAL

// Emisor
Contador_Emisor (CU:= POU_Edges.Rasing_edge_emisor.Q,RESET:= GVL.Reset);
GVL.Contador_Piezas_Totales_Emitidas := WORD_TO_INT(Contador_Emisor.CV);

// Zona Pivot tumbar piezas
Contador_Zona_Pivot (CU:= POU_Edges.Rasing_edge_emisor.Q,CD := POU_Edges.Falling_edge_Limpiador.Q,RESET:= GVL.Reset);
GVL.Contador_Piezas_Zona_Pivot_Principal := WORD_TO_INT(Contador_Zona_Pivot.CV);

// Linea Principal
Contador_Piezas_Descartadas_Totales ( CU:= POU_Edges.Falling_Edge_Descartadas.Q,RESET:= GVL.Reset);
GVL.Contador_Piezas_Totales_Descartadas := WORD_TO_INT(Contador_Piezas_Descartadas_Totales.CV);

Contador_Linea_Principal(CU:= POU_Edges.Rasing_Edge_Limpiador.Q,CD := POU_Edges.Falling_Edge_Descartadas.Q OR POU_Edges.Falling_Edge_Azul_Separada.Q OR POU_Edges.Falling_Edge_Verde_Separada.Q OR POU_Edges.Falling_Edge_Metal_Separada.Q ,RESET:= GVL.Reset);
GVL.Contador_Linea_Principal := WORD_TO_INT(Contador_Linea_Principal.CV);


// Zona Push Azul
Contador_Azul (CU:= POU_Edges.Falling_edge_azul_separada.Q,RESET:= GVL.Reset);
GVL.Contador_Totales_Azul_Separadas := WORD_TO_INT(Contador_Azul.CV);

//Zona Push Verde
Contador_Verde (CU:= POU_Edges.Falling_edge_verde_separada.Q,RESET:= GVL.Reset);
GVL.Contador_Totales_Verde_Separadas := WORD_TO_INT(Contador_Verde.CV);

// Zona Entrada Metal
Contador_Metal (CU:= POU_Edges.Falling_edge_metal_separada.Q,RESET:= GVL.Reset);
GVL.Contador_Totales_Metal_Separadas := WORD_TO_INT(Contador_Metal.CV);


//LINEA AZUL

// Zona Pivot
Contador_Pivot_Azul (CU:= POU_Edges.Falling_edge_azul_separada.Q,CD := POU_Edges.Falling_Edge_Diff_6.Q OR POU_Edges.Falling_Edge_Diff_7.Q,RESET:= GVL.Reset);
GVL.Contador_Pivot_Azul := WORD_TO_INT(Contador_Pivot_Azul.CV);

// Zona Manipuladores 1 y 2
Contador_Linea_Manipulador_1_I (CU:= POU_Edges.Rasing_Edge_Diff_6.Q,CD := POU_Edges.Falling_edge_entrada_manipulador_1.Q,RESET:= GVL.Reset);
GVL.Contador_Linea_Manipulador_1_I := WORD_TO_INT(Contador_Linea_Manipulador_1_I.CV);

Contador_Linea_Manipulador_2_I (CU:= POU_Edges.Rasing_Edge_Diff_7.Q,CD := POU_Edges.Falling_edge_entrada_manipulador_2.Q,RESET:= GVL.Reset);
GVL.Contador_Linea_Manipulador_2_I := WORD_TO_INT(Contador_Linea_Manipulador_2_I.CV);

Contador_Manipulador_1 (CU:= POU_Edges.Falling_edge_entrada_manipulador_1.Q,CD := POU_Edges.rasing_edge_salida_manipulador_1.Q,RESET:= GVL.Reset);
GVL.Contador_Manipulador_1 := WORD_TO_INT(Contador_Manipulador_1.CV);

Contador_Manipulador_2 (CU:= POU_Edges.Falling_edge_entrada_manipulador_2.Q,CD := POU_Edges.rasing_edge_salida_manipulador_2.Q,RESET:= GVL.Reset);
GVL.Contador_Manipulador_2 := WORD_TO_INT(Contador_Manipulador_2.CV);

// Zona Paletizador Azul
Contador_Palets_Azules (CU:= POU_Edges.Falling_edge_Paletizador_1.Q,CD := POU_Edges.Falling_edge_Cruce_1_I.Q,RESET:= GVL.Reset);
GVL.Contador_Palets_Azules := WORD_TO_INT(Contador_Palets_Azules.CV);

Contador_Palets_Azules_Totales (CU:= POU_Edges.Falling_edge_Paletizador_1.Q,RESET:= GVL.Reset);
GVL.Contador_Palets_Azules_Totales := WORD_TO_INT(Contador_Palets_Azules_Totales.CV);


//LINEA VERDE

// Zona Pivot
Contador_Pivot_Verde (CU:= POU_Edges.Falling_edge_verde_separada.Q,CD := POU_Edges.Falling_Edge_Diff_10.Q OR POU_Edges.Falling_Edge_Diff_11.Q,RESET:= GVL.Reset);
GVL.Contador_Pivot_Verde := WORD_TO_INT(Contador_Pivot_Verde.CV);

// Zona Manipuladores 3 y 4
Contador_Linea_Manipulador_3_I (CU:= POU_Edges.Rasing_Edge_Diff_11.Q,CD := POU_Edges.Falling_edge_entrada_manipulador_3.Q,RESET:= GVL.Reset);
GVL.Contador_Linea_Manipulador_3_I := WORD_TO_INT(Contador_Linea_Manipulador_3_I.CV);

Contador_Linea_Manipulador_4_I (CU:= POU_Edges.Rasing_Edge_Diff_10.Q,CD := POU_Edges.Falling_edge_entrada_manipulador_4.Q,RESET:= GVL.Reset);
GVL.Contador_Linea_Manipulador_4_I := WORD_TO_INT(Contador_Linea_Manipulador_4_I.CV);

Contador_Manipulador_3 (CU:= POU_Edges.Falling_edge_entrada_manipulador_3.Q,CD := POU_Edges.Rasing_edge_salida_manipulador_3.Q,RESET:= GVL.Reset);
GVL.Contador_Manipulador_3 := WORD_TO_INT(Contador_Manipulador_3.CV);

Contador_Manipulador_4 (CU:= POU_Edges.Falling_edge_entrada_manipulador_4.Q,CD := POU_Edges.Rasing_edge_salida_manipulador_4.Q,RESET:= GVL.Reset);
GVL.Contador_Manipulador_4 := WORD_TO_INT(Contador_Manipulador_4.CV);

// Zona Paletizador Verde
Contador_Palets_Verdes(CU:= POU_Edges.Falling_edge_Paletizador_2.Q,CD := POU_Edges.Falling_edge_Cruce_1_F.Q,RESET:= GVL.Reset);
GVL.Contador_Palets_Verdes := WORD_TO_INT(Contador_Palets_Verdes.CV);

Contador_Palets_Verdes_Totales (CU:= POU_Edges.Falling_edge_Paletizador_2.Q,RESET:= Reset);
GVL.Contador_Palets_Verdes_Totales := WORD_TO_INT(Contador_Palets_Verdes_Totales.CV);

// Zona cruce
Contador_Linea_Cruce_1 (CU:= POU_Edges.Falling_Edge_Cruce_1_Salida.Q,CD := POU_Edges.Falling_edge_Cruce_2_I.Q,RESET:= GVL.Reset);
GVL.Contador_Linea_Cruce_1 := WORD_TO_INT(Contador_Linea_Cruce_1.CV);


//LINEA METAL

// Zona Pivot

Contador_Pivot_Metal (CU:= POU_Edges.Falling_edge_metal_separada.Q,CD := POU_Edges.Falling_Edge_Diff_13.Q OR POU_Edges.Falling_Edge_Diff_14.Q,RESET:= GVL.Reset);
GVL.Contador_Pivot_Metal := WORD_TO_INT(Contador_Pivot_Metal.CV);

// Zona Manipuladores 5 y 6
Contador_Linea_Manipulador_5_I (CU:= POU_Edges.Rasing_Edge_Diff_14.Q,CD := POU_Edges.Falling_edge_entrada_manipulador_5.Q,RESET:= GVL.Reset);
GVL.Contador_Linea_Manipulador_5_I := WORD_TO_INT(Contador_Linea_Manipulador_5_I.CV);

Contador_Linea_Manipulador_6_I (CU:= POU_Edges.Rasing_Edge_Diff_13.Q,CD := POU_Edges.Falling_edge_entrada_manipulador_6.Q,RESET:= GVL.Reset);
GVL.Contador_Linea_Manipulador_6_I := WORD_TO_INT(Contador_Linea_Manipulador_6_I.CV);

Contador_Manipulador_5 (CU:= POU_Edges.Falling_edge_entrada_manipulador_5.Q,CD := POU_Edges.Rasing_edge_salida_manipulador_5.Q,RESET:= GVL.Reset);
GVL.Contador_Manipulador_5 := WORD_TO_INT(Contador_Manipulador_5.CV);

Contador_Manipulador_6 (CU:= POU_Edges.Falling_edge_entrada_manipulador_6.Q,CD := POU_Edges.Rasing_edge_salida_manipulador_6.Q,RESET:= GVL.Reset);
GVL.Contador_Manipulador_6 := WORD_TO_INT(Contador_Manipulador_6.CV);

// Zona Paletizador Metal
Contador_Palets_Metales_Totales (CU:= POU_Edges.Falling_edge_Paletizador_3.Q,RESET:= GVL.Reset);
GVL.Contador_Palets_Metales_Totales := WORD_TO_INT(Contador_Palets_Metales_Totales.CV);

// Zona cruce
Contador_Linea_Cruce_2 (CU:= POU_Edges.Falling_Edge_Cruce_2_Salida.Q,CD := POU_Edges.Falling_Edge_Almacen_I_D.Q,RESET:= GVL.Reset);
GVL.Contador_Linea_Cruce_2 := WORD_TO_INT(Contador_Linea_Cruce_2.CV);


// ALMACEN
Pallets_Almacenados (CU:= POU_Edges.Falling_Edge_Almacen_I_D.Q,RESET:= GVL.Reset);
GVL.Pallets_Almacenados := WORD_TO_INT(Pallets_Almacenados.CV);

Pallet_Almacen_O (CU:= POU_Edges.Rasing_Edge_Almacen_O.Q,CD := POU_Edges.Falling_Edge_Almacen_O.Q,RESET:= GVL.Reset);
//Pallet_Almacen_O_INT := WORD_TO_INT(Pallet_Almacen_O.CV);

Pallets_Almacenados_Retirados (CU:= POU_Edges.Falling_Edge_Almacen_O.Q,RESET:= GVL.Reset);
GVL.Pallets_Almacenados_Retirados := WORD_TO_INT(Pallets_Almacenados_Retirados.CV);


// ---------------------------------------------------------------- CONTROL DE CINTAS ----------------------------------------------------------------

// TENGO QUE TRASLADAR LAS CINTAS DEL PRINCIPIO DE LA LINEA DE PRODUCCION A LA FUNCIÓN

	// Linea principal
	GVL.Belt_Conveyor_4m_1 := Contador_Piezas_Zona_Pivot_Principal >0 AND Contador_Piezas_Zona_Pivot_Principal <3;   
	GVL.Belt_Conveyor_6m_1 := GVL.Contador_Linea_Principal>0 AND GVL.Contador_Linea_Principal<7 ;
	GVL.Belt_Conveyor_6m_4 := GVL.Belt_Conveyor_6m_1;
	GVL.Belt_Conveyor_6m_5 := GVL.Belt_Conveyor_6m_1;

	// Comienzo Linea Azul
	GVL.Belt_Conveyor_2m_3 := GVL.Contador_Pivot_Azul>0 AND GVL.Contador_Pivot_Azul<3;
	GVL.Belt_Conveyor_2m_4 := GVL.Contador_Pivot_Azul>0;
	GVL.Curved_Belt_Conveyor_1_CW := GVL.Belt_Conveyor_2m_3;
	GVL.Pivot_Arm_Sorter_2_Belt_mas := GVL.Belt_Conveyor_2m_4;
	 
	// Comienzo Linea Verde
	GVL.Belt_Conveyor_2m_7 := GVL.Contador_Pivot_Verde>0 AND GVL.Contador_Pivot_Verde<3;
	GVL.Belt_Conveyor_2m_8 := GVL.Contador_Pivot_Verde>0 ;
	GVL.Curved_Belt_Conveyor_2_CCW := GVL.Belt_Conveyor_2m_7;
	GVL.Pivot_Arm_Sorter_3_Belt_mas := GVL.Belt_Conveyor_2m_8;

	// Comienzo Linea Metal
	GVL.Belt_Conveyor_2m_2 := GVL.Contador_Pivot_Metal>0 AND GVL.Contador_Pivot_Metal<3;
	GVL.Belt_Conveyor_4m_3 := GVL.Contador_Pivot_Metal>0;
	GVL.Curved_Belt_Conveyor_3_CCW := GVL.Belt_Conveyor_2m_2;
	GVL.Pivot_Arm_Sorter_4_Belt_mas := GVL.Belt_Conveyor_4m_3;

	// Entrada Manipuladores Azules
	GVL.Belt_Conveyor_2m_6 := GVL.Contador_Linea_Manipulador_1_I>0 ;	
	GVL.Belt_Conveyor_2m_5 := GVL.Contador_Linea_Manipulador_2_I>0 AND GVL.Contador_Linea_Manipulador_2_I<2;
	GVL.Belt_Conveyor_6m_2 := GVL.Contador_Linea_Manipulador_1_I>0 AND GVL.Contador_Linea_Manipulador_1_I<5;
	GVL.Curved_Belt_Conveyor_1_CCW := GVL.Belt_Conveyor_6m_2;
	
	// Entrada Manipuladores Verdes	
	GVL.Belt_Conveyor_2m_9 := GVL.Contador_Linea_Manipulador_3_I>0 AND GVL.Contador_Linea_Manipulador_3_I<2;	
	GVL.Belt_Conveyor_2m_10 := GVL.Contador_Linea_Manipulador_4_I>0;
	GVL.Belt_Conveyor_6m_3 := GVL.Contador_Linea_Manipulador_4_I>0 AND GVL.Contador_Linea_Manipulador_3_I<5;
	GVL.Curved_Belt_Conveyor_2_CW := GVL.Belt_Conveyor_6m_3;
	
	// Entrada Manipuladores Metales
	GVL.Belt_Conveyor_2m_11 := GVL.Contador_Linea_Manipulador_5_I>0 AND GVL.Contador_Linea_Manipulador_5_I<2;		
	GVL.Belt_Conveyor_2m_12 := GVL.Contador_Linea_Manipulador_6_I>0;
	GVL.Belt_Conveyor_6m_6 := GVL.Contador_Linea_Manipulador_6_I>0 AND GVL.Contador_Linea_Manipulador_5_I<5;
	GVL.Curved_Belt_Conveyor_3_CW :=GVL.Belt_Conveyor_6m_6;
	
	// Comienzo Linea Rodillos
	 // Hay una caja esperando para salir y la linea todavía acepta Palets	
	GVL.Roller_Conveyor_2m_2 := GVL.Sacar_Palet_1 OR (GVL.Contador_Palets_Azules>0 AND GVL.Contador_Palets_Azules<4);
	GVL.Curved_Roller_Conveyor_1_CCW := GVL.Contador_Palets_Azules>0 AND GVL.Contador_Palets_Azules<4;
	GVL.Roller_Conveyor_6m_1 := GVL.Curved_Roller_Conveyor_1_CCW;
	GVL.Chain_Transfer_1_mas := GVL.Curved_Roller_Conveyor_1_CCW;
	
	// Linea salida Paletizador 2
	GVL.Linea_Salida_Libre_2 := GVL.Sacar_Palet_2 AND GVL.Contador_Palets_Verdes=0; 
	
	// Linea Rodillos entre cruces
	GVL.Roller_Conveyor_6m_2 := GVL.Contador_Linea_Cruce_1 >0 AND GVL.Contador_Linea_Cruce_1 <5;
	GVL.Roller_Conveyor_4m_2 := GVL.Contador_Linea_Cruce_1 >0 AND GVL.Contador_Linea_Cruce_1 <4;

	// Linea salida Paletizador 3
	GVL.Linea_Salida_Libre_3 := GVL.Sacar_Palet_3 AND GVL.Contador_Palets_Metal=0; 
	
	// Linea Rodillos entre cruce y almacen
	GVL.Curved_Roller_Conveyor_2_CW := GVL.Contador_Linea_Cruce_2>0 AND GVL.Contador_Linea_Cruce_2<3;
	GVL.Roller_Conveyor_4m_3 := GVL.Curved_Roller_Conveyor_2_CW; 	
	
	GVL.Loading_Conveyor_2 := WORD_TO_INT(Pallet_Almacen_O.CV)>0;
	GVL.Roller_Conveyor_2m_9 := GVL.Loading_Conveyor_2;

END_PROGRAM

// ---- POUs/Control funcionalidad/FB_Control_Estacion.TcPOU
FUNCTION_BLOCK FB_Control_Estacion
VAR_INPUT
	Start_Button : BOOL;
	Stop_Button : BOOL;
	Reset_Button : BOOL;
	Safety_Door : BOOL;
	
END_VAR
VAR_IN_OUT
	Estado             : INT;
END_VAR
VAR_OUTPUT
	Control 		   : BOOL;
	Start_Button_Light : BOOL;
	Stop_Button_Light  : BOOL;
	Reset_Button_Light : BOOL;
	Stack_Light_Green  : BOOL;	 
	Stack_Light_Red    : BOOL;	
	Stack_Light_Yellow : BOOL;
	
END_VAR
VAR	
END_VAR

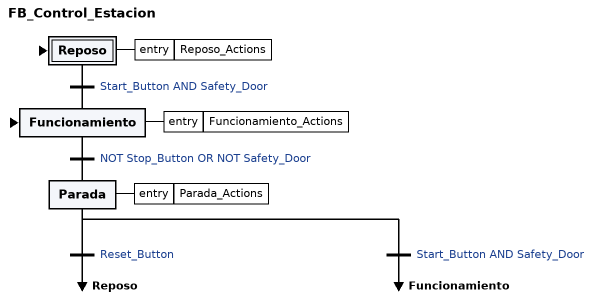
INITIAL_STEP Reposo:
    Reposo_Actions(P1);  // entry action
END_STEP
TRANSITION FROM Reposo TO Funcionamiento
    := Start_Button AND Safety_Door;
END_TRANSITION
STEP Funcionamiento:
    Funcionamiento_Actions(P1);  // entry action
END_STEP
TRANSITION FROM Funcionamiento TO Parada
    := NOT Stop_Button OR NOT Safety_Door;
END_TRANSITION
STEP Parada:
    Parada_Actions(P1);  // entry action
END_STEP
TRANSITION FROM Parada TO Reposo
    := Reset_Button;
END_TRANSITION
TRANSITION FROM Parada TO Funcionamiento
    := Start_Button AND Safety_Door;
END_TRANSITION

ACTION Funcionamiento_Actions:
Control := TRUE; // Se indica que la estación puede funcionar
// Se indica mediante una luz que el siguiente botón a pulsar sería el de Stop
Start_Button_Light := FALSE;
Stop_Button_Light := TRUE;
Reset_Button_Light := FALSE;
//Semáforo indicando estación en funcionamiento
Stack_Light_Green := TRUE; 
Stack_Light_Red := FALSE;	
Stack_Light_Yellow := FALSE;
END_ACTION

ACTION Parada_Actions:
Control := FALSE; // Se indica que la estación no puede funcionar
// Se indica mediante una luz que el siguiente botón a pulsar sería el de Stop o el reset dependiendo de la acción deseada
Stop_Button_Light := FALSE;
Start_Button_Light := TRUE;
Reset_Button_Light := TRUE;
//Semáforo indicando que se ha solicitado la parada de la estación
Stack_Light_Green := FALSE;
Stack_Light_Red := FALSE;	
Stack_Light_Yellow := TRUE;
END_ACTION

ACTION Reposo_Actions:
Control := FALSE; // Se indica que la planta no puede funcionar
// Se indica mediante una luz que el siguiente botón a pulsar sería el de Start
Start_Button_Light := TRUE;
Stop_Button_Light := FALSE;
Reset_Button_Light := FALSE;
Estado := 0;
//Semáforo indicando estación parada
Stack_Light_Green := FALSE;	 
Stack_Light_Red := TRUE;	
Stack_Light_Yellow := FALSE;
END_ACTION

END_FUNCTION_BLOCK

// ---- POUs/Control funcionalidad/POU_Reset_Planta.TcPOU
PROGRAM POU_Reset_Planta
VAR
	i : INT ;
END_VAR

	GVL.Reset := TRUE;

	// VARIABLES PARA CONTROLAR ACCIONES	
	
	GVL.Control_TAPP_A 			 := FALSE; // En base a la botonera de control y los sensores de puerta, se permite el movimiento o no
	GVL.Control_TAPP_V 			 := FALSE; // En base a la botonera de control y los sensores de puerta, se permite el movimiento o no
	GVL.Control_TAPP_M 			 := FALSE; // En base a la botonera de control y los sensores de puerta, se permite el movimiento o no
	GVL.Control_Paletizador_A 	 := FALSE; // En base a la botonera de control y los sensores de puerta, se permite el movimiento o no
	GVL.Control_Paletizador_V 	 := FALSE; // En base a la botonera de control y los sensores de puerta, se permite el movimiento o no
	GVL.Control_Paletizador_M 	 := FALSE; // En base a la botonera de control y los sensores de puerta, se permite el movimiento o no
	GVL.Control_Almacen 	 := FALSE; // En base a la botonera de control y los sensores de puerta, se permite el movimiento o no		
	GVL.Error_RFID_1  := FALSE; // Variable que guarda si ha habido error a la hora de escribir información en un palet	
	GVL.Error_RFID_2  := FALSE; // Variable que guarda si ha habido error a la hora de escribir información en un palet	
	GVL.Error_RFID_3  := FALSE; // Variable que guarda si ha habido error a la hora de escribir información en un palet
	GVL.Error_RFID_Almacen  := FALSE; // Variable que guarda si ha habido error a la hora de leer información en un palet	
	GVL.Linea_Salida_Libre_2  := TRUE; // Control de cinta de salida para el paletizado, si la línea de salida no está libre, no puede sacar el palet
	GVL.Linea_Salida_Libre_3  := TRUE; // Control de cinta de salida para el paletizado, si la línea de salida no está libre, no puede sacar el palet
	GVL.Sacar_Palet_1  := FALSE; // Para saber si el palet del paletizador tiene via libre para ser pasado a los rodillos camino al almacen
	GVL.Sacar_Palet_2  := FALSE; // Para saber si el palet del paletizador tiene via libre para ser pasado a los rodillos camino al almacen
	GVL.Sacar_Palet_3  := FALSE; // Para saber si el palet del paletizador tiene via libre para ser pasado a los rodillos camino al almacen
	
	//ESTADOS	
	GVL.Estado_Pick_Place_1 	  := 0;
	GVL.Estado_Palletizer_1 	  := 0;
	GVL.Estado_Pick_Place_2 	  := 0;
	GVL.Estado_Palletizer_2 	  := 0;
	GVL.Estado_Pick_Place_3 	  := 0;
	GVL.Estado_Palletizer_3 	  := 0;	
	GVL.Estado_Almacen_I 	 	:= 0; // Almacenar un palet en el almacen
	GVL.Estado_Almacen_O 	 	:= 1; // Extraer un palet del almacen
	
	// ALMACEN
	
	GVL.ContadorPalets			 := 0; // Contador de palets del Almacen en base a la selección del display
	GVL.Retirada_Start			 := FALSE; // Guarda la pulsación del botón start para extraer del almacen
	GVL.Reset := FALSE;

END_PROGRAM

// ---- POUs/Entrada y división/Etapa1.TcPOU
FUNCTION_BLOCK Etapa1
VAR_INPUT
END_VAR
VAR_OUTPUT
END_VAR
VAR
	
	//Accionar_Push_1 				: BOOL 	:= FALSE;	
	Contador_Linea_Principal 		: INT 	:= -1; // piezas que han entrado en la línea principal
	Contador_Sensor_Zona_Metal 		: INT 	:= 0; // piezas que pasan por el sensor de la linea metálica
	Contador_Sensor_Zona_Verde 		: INT 	:= 0; // piezas que pasan por el sensor de la linea verde
	Posicion_Array_Azul 			: INT 	:= -1; // posición a consultar para accionar el pusher azul	
	Pieza 							: DINT 	:= 0; // Tipo de elemento que pasa por el sensor de vision
	Piezas_Entrada 					: ARRAY[0..4] OF DINT := [4(0)]; // array que guarda la información de los elementos que hay entre el pusher 1 y 2
	Piezas_Zona_Metal				: ARRAY[0..10] OF DINT := [10(0)]; // array que guarda la información de los elementos que hay entre el pusher 2 y 3
	Posicion_Array_Metal			: INT 	:= 0; // posición a consultar para accionar el pusher verde	
	Posicion_Array_Verde			: INT 	:= 0; // posición a consultar para accionar el pusher metálico	
		
END_VAR

// ---------------------------------------------------------------- 1. PIVOT ARM ENTRADA ----------------------------------------------------------------

// Control para tumbar las piezas. Esta parte funcionará si hay piezas en la cinta. Dependiendo de la orientación y posición, es posible que el objeto se quede "estancado" debajo del Pivot, este caso se
// reconocerá cuando los sensores de entrada y salida detecten objetos a la vez, ya que el tiempo de emisión está diseñado para que no tengan que coincidir. Cuando esto sucede, de invertirá el 
// sentido de giro para "desatascar" la pieza. En caso contrario, se mantiene el giro predefinido.

 GVL.Pivot_Arm_Sorter_1_Belt_mas := GVL.Contador_Piezas_Zona_Pivot_Principal >0 AND NOT ( GVL.Diffuse_Sensor_0 AND GVL.Diffuse_Sensor_1);
 GVL.Pivot_Arm_Sorter_1_Belt_menos := GVL.Contador_Piezas_Zona_Pivot_Principal >0 AND GVL.Diffuse_Sensor_0 AND GVL.Diffuse_Sensor_1;

// ---------------------------------------------------------------- 2. CONTROL DESCARTE Y RELLENO DEL ARRAY----------------------------------------------------------------
 
// Si las líneas de entrada no aceptan más piezas, se descartan las pezas de color
IF GVL.Contador_Pivot_Azul>=3 THEN GVL.Input[0].Descartar_Pieza_Azul := TRUE; ELSE GVL.Input[0].Descartar_Pieza_Azul := FALSE; END_IF
IF GVL.Contador_Pivot_Verde>=3 THEN GVL.Input[0].Descartar_Pieza_Verde := TRUE; ELSE GVL.Input[0].Descartar_Pieza_Verde := FALSE; END_IF
IF GVL.Contador_Pivot_Metal>=3 THEN GVL.Input[0].Descartar_Pieza_Metal := TRUE; ELSE GVL.Input[0].Descartar_Pieza_Metal := FALSE; END_IF

// Control para descartar las piezas: he tenido que meter un control porque dependiendo de la longitud, el sensor deja de leer antes de que 
//la pieza acabe de pasar ya que lee en el centro de la pieza y si esta es muy larga el centro sale antes de que acabe de salir la pieza  
IF POU_Edges.Rasing_Edge_Sensor_Zona_Azul.Q THEN 
	Contador_Linea_Principal:=Contador_Linea_Principal+1;
	Piezas_Entrada[Contador_Linea_Principal MOD 4]:= GVL.Vision_Sensor_1; ;	
END_IF

// ---------------------------------------------------------------- 3. PUSHER AZUL ----------------------------------------------------------------
//El push se acciona si la pieza que tiene colocada delante es azul
IF POU_Edges.Falling_edge_sensor_zona_azul.Q THEN
	Posicion_Array_Azul:=Posicion_Array_Azul+1;
	IF Piezas_Entrada[Posicion_Array_Azul MOD 4] = 1 AND NOT GVL.Input[0].Descartar_Pieza_Azul THEN 
		GVL.Pusher_1 := TRUE;
	END_IF
END_IF
    
IF GVL.Pusher_1_Front_Limit THEN GVL.Pusher_1 := FALSE; END_IF

// ---------------------------------------------------------------- 4. PUSHER VERDE----------------------------------------------------------------
//El push se acciona si la pieza que tiene colocada delante es verde
IF POU_Edges.Falling_edge_sensor_zona_verde.Q THEN
	  Contador_Sensor_Zona_Verde := Contador_Sensor_Zona_Verde+1;	
	  Posicion_Array_Verde := Contador_Sensor_Zona_Verde + GVL.Contador_Totales_Azul_Separadas;
	  Posicion_Array_Metal := Contador_Sensor_Zona_Verde - GVL.Contador_Totales_Verde_Separadas;
	IF Piezas_Entrada[(Posicion_Array_Verde-1)MOD 4] = 4 AND NOT GVL.Input[0].Descartar_Pieza_Verde THEN 
		GVL.Pusher_2 := TRUE;
	ELSE Piezas_Zona_Metal [(Posicion_Array_Metal-1) MOD 10] := Piezas_Entrada[(Posicion_Array_Verde-1)MOD 4]; // Si la pieza no es verde, de envia el valor al array destinado al push para piezas metálicas
	END_IF
END_IF
    
IF GVL.Pusher_2_Front_Limit THEN GVL.Pusher_2 := FALSE; END_IF

// ---------------------------------------------------------------- 5. PUSHER METAL----------------------------------------------------------------
//El push se acciona si la pieza que tiene colocada delante es verde
IF POU_Edges.Falling_edge_sensor_zona_metal.Q THEN
		Contador_Sensor_Zona_Metal := Contador_Sensor_Zona_Metal+1;
	IF Piezas_Zona_Metal[(Contador_Sensor_Zona_Metal-1) MOD 10] = 7 AND NOT GVL.Input[0].Descartar_Pieza_Metal THEN 
		GVL.Pusher_3 := TRUE;
	END_IF
	
END_IF
    
IF GVL.Pusher_3_Front_Limit THEN GVL.Pusher_3 := FALSE; END_IF

END_FUNCTION_BLOCK

// ---- POUs/Línea producción/POU_Pinzas.TcPOU
FUNCTION_BLOCK POU_Pinzas
VAR_INPUT
	Falling_Edge_Entrada_Pinza 	: BOOL;
	Falling_Edge_Salida_Pinza 	: BOOL;
	Right_Positioner_Clamped 	: BOOL;
END_VAR
VAR_OUTPUT
	Emitter_Box					: BOOL;
	Right_Positioner_Clamp 		: BOOL;
	Right_Positioner_Raise 		: BOOL;	
END_VAR
VAR_IN_OUT
	Cinta_Libre 				: BOOL;
	Contador_Manipulador_Base 	: INT;
	Contador_Box 				: INT;	
	Hay_Pieza 					: WSTRING ;
END_VAR

// ACCIONES PINZA 2

// muevo la cinta si no hay pieza en el posicionador
// Si entra una pieza al posicionador, cierro la pinza y paro la cinta
IF Falling_Edge_Entrada_Pinza THEN 
	Right_Positioner_Clamp := TRUE;
	Cinta_Libre := FALSE;
	
END_IF

// Una vez cerrada la pinza vuelvo a abrirla
IF Right_Positioner_Clamped THEN
	
	Right_Positioner_Clamp := FALSE;
	Hay_Pieza := "Base";
	
END_IF

// Si hay pieza soldada levanto la pinza
IF Hay_Pieza = "Completa" THEN
	
	Right_Positioner_Raise:=TRUE;
	Cinta_Libre := TRUE;
	Hay_Pieza := "Vacio";	
	
END_IF

Emitter_Box := Falling_Edge_Salida_Pinza;
	
// Una vez la pieza haya pasado el clamp, lo bajamos para posicionar la siguiente pieza
IF Falling_Edge_Salida_Pinza THEN
	
	Right_Positioner_Raise := FALSE;	
	Contador_Manipulador_Base := Contador_Manipulador_Base-1;
	Contador_Box := Contador_Box +1;
	
END_IF

END_FUNCTION_BLOCK

// ---- POUs/Módulos/POU_Mando.TcPOU
PROGRAM POU_Mando
VAR
END_VAR

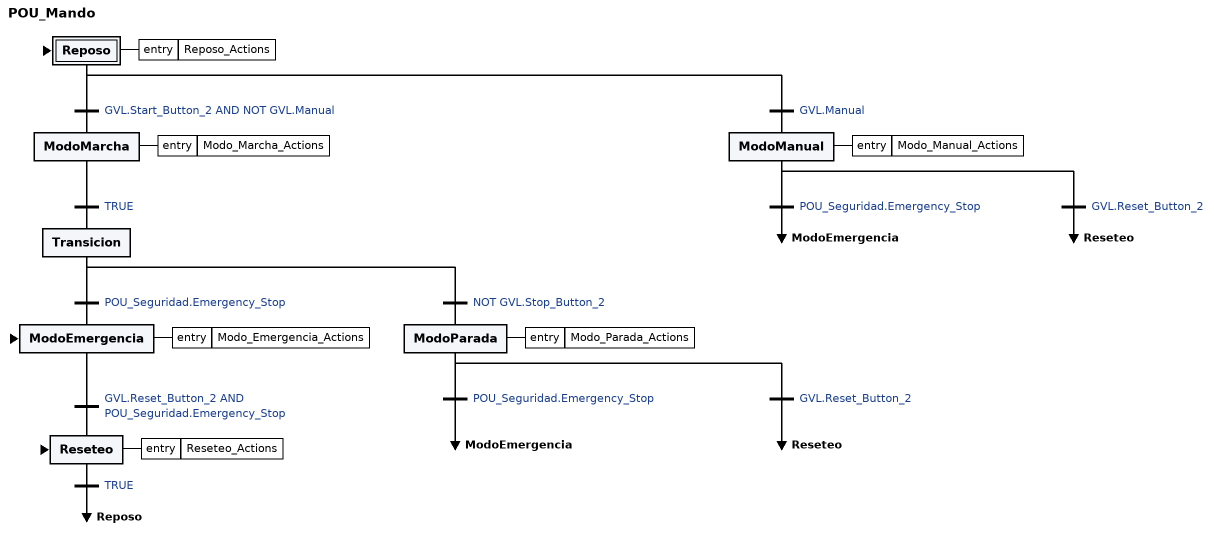
INITIAL_STEP Reposo:
    Reposo_Actions(P1);  // entry action
END_STEP
TRANSITION FROM Reposo TO ModoMarcha
    := GVL.Start_Button_2 AND NOT GVL.Manual;
END_TRANSITION
STEP ModoMarcha:
    Modo_Marcha_Actions(P1);  // entry action
END_STEP
TRANSITION FROM ModoMarcha TO Transicion
    := TRUE;
END_TRANSITION
TRANSITION FROM Reposo TO ModoManual
    := GVL.Manual;
END_TRANSITION
STEP ModoManual:
    Modo_Manual_Actions(P1);  // entry action
END_STEP
TRANSITION FROM ModoManual TO ModoEmergencia
    := POU_Seguridad.Emergency_Stop;
END_TRANSITION
TRANSITION FROM ModoManual TO Reseteo
    := GVL.Reset_Button_2;
END_TRANSITION
STEP Transicion:
END_STEP
TRANSITION FROM Transicion TO ModoEmergencia
    := POU_Seguridad.Emergency_Stop;
END_TRANSITION
STEP ModoEmergencia:
    Modo_Emergencia_Actions(P1);  // entry action
END_STEP
TRANSITION FROM ModoEmergencia TO Reseteo
    := GVL.Reset_Button_2 AND POU_Seguridad.Emergency_Stop;
END_TRANSITION
TRANSITION FROM Transicion TO ModoParada
    := NOT GVL.Stop_Button_2;
END_TRANSITION
STEP ModoParada:
    Modo_Parada_Actions(P1);  // entry action
END_STEP
TRANSITION FROM ModoParada TO ModoEmergencia
    := POU_Seguridad.Emergency_Stop;
END_TRANSITION
TRANSITION FROM ModoParada TO Reseteo
    := GVL.Reset_Button_2;
END_TRANSITION
STEP Reseteo:
    Reseteo_Actions(P1);  // entry action
END_STEP
TRANSITION FROM Reseteo TO Reposo
    := TRUE;
END_TRANSITION

ACTION Desactivar_Alarmas_Actions:
//Se desactivan las alarmas
GVL.Alarm_Siren  := FALSE;
GVL.Warning_Light  := FALSE;
GVL.Factory_IO_Pause := FALSE;
END_ACTION

ACTION Modo_Emergencia_Actions:
GVL.Marcha := FALSE; // Se indica que la planta no puede funcionar
END_ACTION

ACTION Modo_Manual_Actions:
// Se indica mediante una luz que el siguiente botón a pulsar sería el de Reset
GVL.Start_Button_2_Light := FALSE;
GVL.Reset_Button_2_Light := TRUE;
END_ACTION

ACTION Modo_Marcha_Actions:
GVL.Marcha := TRUE; // Se indica que la planta puede comenzar a funcionar
GVL.Emitter_1 := TRUE; // Se activa la emisión de piezas
GVL.Belt_Conveyor_2m_1 := 1; // Se activa la cinta de entrada
// Se indica mediante una luz que el siguiente botón a pulsar sería el de Stop
GVL.Start_Button_2_Light := FALSE; 
GVL.Stop_Button_2_Light := TRUE;
END_ACTION

ACTION Modo_Parada_Actions:
GVL.Emitter_1 := FALSE; // Se desactiva la emisión de piezas
GVL.Belt_Conveyor_2m_1 := 0; // Se desactiva la cinta de entrada
// Se indica mediante una luz que el siguiente botón a pulsar sería el de Reset
GVL.Stop_Button_2_Light := FALSE; 
GVL.Reset_Button_2_Light := TRUE;
END_ACTION

ACTION Reposo_Actions:
GVL.Marcha := FALSE; // Se indica que la planta no puede funcionar
// Se indica mediante una luz que el siguiente botón a pulsar sería el de Start
GVL.Start_Button_2_Light := TRUE; 
GVL.Reset_Button_2_Light := FALSE;
// Se permite que la planta se mueva dentro del factory I/O
GVL.Factory_IO_Pause := FALSE;
GVL.Factory_IO_Reset := FALSE;
END_ACTION

ACTION Reseteo_Actions:
GVL.Factory_IO_Reset := TRUE;
POU_Reset_Planta();
GVL.Manual := FALSE;
//Se desactivan las alarmas
//GVL.Alarm_Siren  := FALSE;
//GVL.Warning_Light  := FALSE;
END_ACTION

END_PROGRAM

// ---- POUs/Módulos/POU_Seguridad.TcPOU
PROGRAM POU_Seguridad
VAR
	Emergency_Stop : BOOL := FALSE; // variable para indicar la parada inmediata de la planta
END_VAR

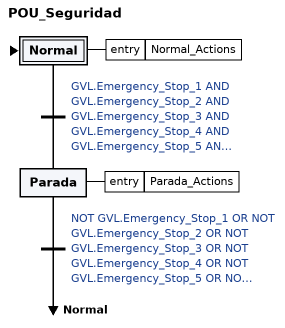
INITIAL_STEP Normal:
    Normal_Actions(P1);  // entry action
END_STEP
TRANSITION FROM Normal TO Parada
    := GVL.Emergency_Stop_1 AND GVL.Emergency_Stop_2 AND GVL.Emergency_Stop_3 AND GVL.Emergency_Stop_4 AND GVL.Emergency_Stop_5 AND GVL.Emergency_Stop_6 AND GVL.Emergency_Stop_7 AND GVL.Emergency_Stop_8 AND GVL.Emergency_Stop_9;
END_TRANSITION
STEP Parada:
    Parada_Actions(P1);  // entry action
END_STEP
TRANSITION FROM Parada TO Normal
    := NOT GVL.Emergency_Stop_1 OR NOT GVL.Emergency_Stop_2 OR NOT GVL.Emergency_Stop_3 OR NOT GVL.Emergency_Stop_4 OR NOT GVL.Emergency_Stop_5 OR NOT GVL.Emergency_Stop_6 OR NOT GVL.Emergency_Stop_7 OR NOT GVL.Emergency_Stop_8 OR NOT GVL.Emergency_Stop_9;
END_TRANSITION

ACTION Normal_Actions:
 Emergency_Stop := FALSE;
 //Se desactivan las alarmas
GVL.Alarm_Siren  := FALSE;
GVL.Warning_Light  := FALSE;
GVL.Factory_IO_Pause := FALSE;
END_ACTION

ACTION Parada_Actions:
 Emergency_Stop := TRUE;
 // Se indica mediante una luz que el siguiente botón a pulsar sería el de Reset
GVL.Stop_Button_2_Light := FALSE;
GVL.Reset_Button_2_Light := TRUE;
//Se activan las alarmas
GVL.Alarm_Siren  := TRUE;
GVL.Warning_Light  := TRUE;
POU_Parada();
END_ACTION

END_PROGRAM

